    CONST robtarget T2024:=[[60.250034,78.904563,16.249831],[1.000000,0.000000,0.000000,0.000000],[0,0,-1,0],[9E+09,9E+09,9E+09,9E+09,9E+09,9E+09]];
    CONST robtarget T2025:=[[60.250034,32.487797,16.249831],[1.000000,0.000000,0.000000,0.000000],[0,0,-1,0],[9E+09,9E+09,9E+09,9E+09,9E+09,9E+09]];
    CONST robtarget T2026:=[[61.750040,32.676352,16.249831],[1.000000,0.000000,0.000000,0.000000],[0,0,-1,0],[9E+09,9E+09,9E+09,9E+09,9E+09,9E+09]];
    CONST robtarget T2027:=[[61.750040,78.498231,16.249831],[1.000000,0.000000,0.000000,0.000000],[0,0,-1,0],[9E+09,9E+09,9E+09,9E+09,9E+09,9E+09]];
    CONST robtarget T2028:=[[63.250046,77.962337,16.249831],[1.000000,0.000000,0.000000,0.000000],[0,0,-1,0],[9E+09,9E+09,9E+09,9E+09,9E+09,9E+09]];
    CONST robtarget T2029:=[[63.250046,32.936847,16.249831],[1.000000,0.000000,0.000000,0.000000],[0,0,-1,0],[9E+09,9E+09,9E+09,9E+09,9E+09,9E+09]];
    CONST robtarget T2030:=[[64.750052,33.276223,16.249831],[1.000000,0.000000,0.000000,0.000000],[0,0,-1,0],[9E+09,9E+09,9E+09,9E+09,9E+09,9E+09]];
    CONST robtarget T2031:=[[64.750052,77.237553,16.249831],[1.000000,0.000000,0.000000,0.000000],[0,0,-1,0],[9E+09,9E+09,9E+09,9E+09,9E+09,9E+09]];
    CONST robtarget T2032:=[[66.250058,76.248790,16.249831],[1.000000,0.000000,0.000000,0.000000],[0,0,-1,0],[9E+09,9E+09,9E+09,9E+09,9E+09,9E+09]];
    CONST robtarget T2033:=[[66.250058,33.701895,16.249831],[1.000000,0.000000,0.000000,0.000000],[0,0,-1,0],[9E+09,9E+09,9E+09,9E+09,9E+09,9E+09]];
    CONST robtarget T2034:=[[67.750064,34.280483,16.249831],[1.000000,0.000000,0.000000,0.000000],[0,0,-1,0],[9E+09,9E+09,9E+09,9E+09,9E+09,9E+09]];
    CONST robtarget T2035:=[[67.750064,74.766975,16.249831],[1.000000,0.000000,0.000000,0.000000],[0,0,-1,0],[9E+09,9E+09,9E+09,9E+09,9E+09,9E+09]];
    CONST robtarget T2036:=[[69.250070,72.779272,16.249831],[1.000000,0.000000,0.000000,0.000000],[0,0,-1,0],[9E+09,9E+09,9E+09,9E+09,9E+09,9E+09]];
    CONST robtarget T2037:=[[69.250070,34.893685,16.249831],[1.000000,0.000000,0.000000,0.000000],[0,0,-1,0],[9E+09,9E+09,9E+09,9E+09,9E+09,9E+09]];
    CONST robtarget T2038:=[[70.750076,35.855715,16.249831],[1.000000,0.000000,0.000000,0.000000],[0,0,-1,0],[9E+09,9E+09,9E+09,9E+09,9E+09,9E+09]];
    CONST robtarget T2039:=[[70.750076,70.592401,16.249831],[1.000000,0.000000,0.000000,0.000000],[0,0,-1,0],[9E+09,9E+09,9E+09,9E+09,9E+09,9E+09]];
    CONST robtarget T2040:=[[72.250082,71.487627,16.249831],[1.000000,0.000000,0.000000,0.000000],[0,0,-1,0],[9E+09,9E+09,9E+09,9E+09,9E+09,9E+09]];
    CONST robtarget T2041:=[[72.250082,36.807675,16.249831],[1.000000,0.000000,0.000000,0.000000],[0,0,-1,0],[9E+09,9E+09,9E+09,9E+09,9E+09,9E+09]];
    CONST robtarget T2042:=[[73.750088,38.399045,16.249831],[1.000000,0.000000,0.000000,0.000000],[0,0,-1,0],[9E+09,9E+09,9E+09,9E+09,9E+09,9E+09]];
    CONST robtarget T2043:=[[73.750088,70.448227,16.249831],[1.000000,0.000000,0.000000,0.000000],[0,0,-1,0],[9E+09,9E+09,9E+09,9E+09,9E+09,9E+09]];
    CONST robtarget T2044:=[[75.250094,67.768342,16.249831],[1.000000,0.000000,0.000000,0.000000],[0,0,-1,0],[9E+09,9E+09,9E+09,9E+09,9E+09,9E+09]];
    CONST robtarget T2045:=[[75.250094,40.369976,16.249831],[1.000000,0.000000,0.000000,0.000000],[0,0,-1,0],[9E+09,9E+09,9E+09,9E+09,9E+09,9E+09]];
    CONST robtarget T2046:=[[76.750100,43.140634,16.249831],[1.000000,0.000000,0.000000,0.000000],[0,0,-1,0],[9E+09,9E+09,9E+09,9E+09,9E+09,9E+09]];
    CONST robtarget T2047:=[[76.750100,63.221678,16.249831],[1.000000,0.000000,0.000000,0.000000],[0,0,-1,0],[9E+09,9E+09,9E+09,9E+09,9E+09,9E+09]];
    CONST robtarget T2048:=[[78.250106,56.651419,16.249831],[1.000000,0.000000,0.000000,0.000000],[0,0,-1,0],[9E+09,9E+09,9E+09,9E+09,9E+09,9E+09]];
    CONST robtarget T2049:=[[78.250106,48.862612,16.249831],[1.000000,0.000000,0.000000,0.000000],[0,0,-1,0],[9E+09,9E+09,9E+09,9E+09,9E+09,9E+09]];
    CONST robtarget T2050:=[[77.500103,48.233244,16.749841],[1.000000,0.000000,0.000000,0.000000],[0,0,-1,0],[9E+09,9E+09,9E+09,9E+09,9E+09,9E+09]];
    CONST robtarget T2051:=[[77.500103,59.623165,16.749841],[1.000000,0.000000,0.000000,0.000000],[0,0,-1,0],[9E+09,9E+09,9E+09,9E+09,9E+09,9E+09]];
    CONST robtarget T2052:=[[77.500103,48.233244,16.749841],[1.000000,0.000000,0.000000,0.000000],[0,0,-1,0],[9E+09,9E+09,9E+09,9E+09,9E+09,9E+09]];
    CONST robtarget T2053:=[[77.500103,59.623165,16.749841],[1.000000,0.000000,0.000000,0.000000],[0,0,-1,0],[9E+09,9E+09,9E+09,9E+09,9E+09,9E+09]];
    CONST robtarget T2054:=[[76.000097,65.184856,16.749841],[1.000000,0.000000,0.000000,0.000000],[0,0,-1,0],[9E+09,9E+09,9E+09,9E+09,9E+09,9E+09]];
    CONST robtarget T2055:=[[76.000097,41.932974,16.749841],[1.000000,0.000000,0.000000,0.000000],[0,0,-1,0],[9E+09,9E+09,9E+09,9E+09,9E+09,9E+09]];
    CONST robtarget T2056:=[[74.500091,39.400333,16.749841],[1.000000,0.000000,0.000000,0.000000],[0,0,-1,0],[9E+09,9E+09,9E+09,9E+09,9E+09,9E+09]];
    CONST robtarget T2057:=[[74.500091,69.124433,16.749841],[1.000000,0.000000,0.000000,0.000000],[0,0,-1,0],[9E+09,9E+09,9E+09,9E+09,9E+09,9E+09]];
    CONST robtarget T2058:=[[73.000085,71.338605,16.749841],[1.000000,0.000000,0.000000,0.000000],[0,0,-1,0],[9E+09,9E+09,9E+09,9E+09,9E+09,9E+09]];
    CONST robtarget T2059:=[[73.000085,37.732430,16.749841],[1.000000,0.000000,0.000000,0.000000],[0,0,-1,0],[9E+09,9E+09,9E+09,9E+09,9E+09,9E+09]];
    CONST robtarget T2060:=[[71.500079,36.421505,16.749841],[1.000000,0.000000,0.000000,0.000000],[0,0,-1,0],[9E+09,9E+09,9E+09,9E+09,9E+09,9E+09]];
    CONST robtarget T2061:=[[71.500079,70.991778,16.749841],[1.000000,0.000000,0.000000,0.000000],[0,0,-1,0],[9E+09,9E+09,9E+09,9E+09,9E+09,9E+09]];
    CONST robtarget T2062:=[[70.000073,71.577935,16.749841],[1.000000,0.000000,0.000000,0.000000],[0,0,-1,0],[9E+09,9E+09,9E+09,9E+09,9E+09,9E+09]];
    CONST robtarget T2063:=[[70.000073,35.459476,16.749841],[1.000000,0.000000,0.000000,0.000000],[0,0,-1,0],[9E+09,9E+09,9E+09,9E+09,9E+09,9E+09]];
    CONST robtarget T2064:=[[68.500067,34.636854,16.749841],[1.000000,0.000000,0.000000,0.000000],[0,0,-1,0],[9E+09,9E+09,9E+09,9E+09,9E+09,9E+09]];
    CONST robtarget T2065:=[[68.500067,73.714208,16.749841],[1.000000,0.000000,0.000000,0.000000],[0,0,-1,0],[9E+09,9E+09,9E+09,9E+09,9E+09,9E+09]];
    CONST robtarget T2066:=[[67.000061,75.529975,16.749841],[1.000000,0.000000,0.000000,0.000000],[0,0,-1,0],[9E+09,9E+09,9E+09,9E+09,9E+09,9E+09]];
    CONST robtarget T2067:=[[67.000061,34.067929,16.749841],[1.000000,0.000000,0.000000,0.000000],[0,0,-1,0],[9E+09,9E+09,9E+09,9E+09,9E+09,9E+09]];
    CONST robtarget T2068:=[[65.500055,33.523693,16.749841],[1.000000,0.000000,0.000000,0.000000],[0,0,-1,0],[9E+09,9E+09,9E+09,9E+09,9E+09,9E+09]];
    CONST robtarget T2069:=[[65.500055,76.783651,16.749841],[1.000000,0.000000,0.000000,0.000000],[0,0,-1,0],[9E+09,9E+09,9E+09,9E+09,9E+09,9E+09]];
    CONST robtarget T2070:=[[64.000049,77.607482,16.749841],[1.000000,0.000000,0.000000,0.000000],[0,0,-1,0],[9E+09,9E+09,9E+09,9E+09,9E+09,9E+09]];
    CONST robtarget T2071:=[[64.000049,33.181966,16.749841],[1.000000,0.000000,0.000000,0.000000],[0,0,-1,0],[9E+09,9E+09,9E+09,9E+09,9E+09,9E+09]];
    CONST robtarget T2072:=[[62.500043,32.845958,16.749841],[1.000000,0.000000,0.000000,0.000000],[0,0,-1,0],[9E+09,9E+09,9E+09,9E+09,9E+09,9E+09]];
    CONST robtarget T2073:=[[62.500043,78.210676,16.749841],[1.000000,0.000000,0.000000,0.000000],[0,0,-1,0],[9E+09,9E+09,9E+09,9E+09,9E+09,9E+09]];
    CONST robtarget T2074:=[[61.000037,78.726702,16.749841],[1.000000,0.000000,0.000000,0.000000],[0,0,-1,0],[9E+09,9E+09,9E+09,9E+09,9E+09,9E+09]];
    CONST robtarget T2075:=[[61.000037,32.654827,16.749841],[1.000000,0.000000,0.000000,0.000000],[0,0,-1,0],[9E+09,9E+09,9E+09,9E+09,9E+09,9E+09]];
    CONST robtarget T2076:=[[59.500031,32.472908,16.749841],[1.000000,0.000000,0.000000,0.000000],[0,0,-1,0],[9E+09,9E+09,9E+09,9E+09,9E+09,9E+09]];
    CONST robtarget T2077:=[[59.500031,79.071134,16.749841],[1.000000,0.000000,0.000000,0.000000],[0,0,-1,0],[9E+09,9E+09,9E+09,9E+09,9E+09,9E+09]];
    CONST robtarget T2078:=[[58.000025,79.360542,16.749841],[1.000000,0.000000,0.000000,0.000000],[0,0,-1,0],[9E+09,9E+09,9E+09,9E+09,9E+09,9E+09]];
    CONST robtarget T2079:=[[58.000025,32.352211,16.749841],[1.000000,0.000000,0.000000,0.000000],[0,0,-1,0],[9E+09,9E+09,9E+09,9E+09,9E+09,9E+09]];
    CONST robtarget T2080:=[[56.500019,32.279634,16.749841],[1.000000,0.000000,0.000000,0.000000],[0,0,-1,0],[9E+09,9E+09,9E+09,9E+09,9E+09,9E+09]];
    CONST robtarget T2081:=[[56.500019,79.716007,16.749841],[1.000000,0.000000,0.000000,0.000000],[0,0,-1,0],[9E+09,9E+09,9E+09,9E+09,9E+09,9E+09]];
    CONST robtarget T2082:=[[55.000013,79.976085,16.749841],[1.000000,0.000000,0.000000,0.000000],[0,0,-1,0],[9E+09,9E+09,9E+09,9E+09,9E+09,9E+09]];
    CONST robtarget T2083:=[[55.000013,32.242406,16.749841],[1.000000,0.000000,0.000000,0.000000],[0,0,-1,0],[9E+09,9E+09,9E+09,9E+09,9E+09,9E+09]];
    CONST robtarget T2084:=[[53.500007,32.279634,16.749841],[1.000000,0.000000,0.000000,0.000000],[0,0,-1,0],[9E+09,9E+09,9E+09,9E+09,9E+09,9E+09]];
    CONST robtarget T2085:=[[53.500007,79.716007,16.749841],[1.000000,0.000000,0.000000,0.000000],[0,0,-1,0],[9E+09,9E+09,9E+09,9E+09,9E+09,9E+09]];
    CONST robtarget T2086:=[[52.000001,79.360541,16.749841],[1.000000,0.000000,0.000000,0.000000],[0,0,-1,0],[9E+09,9E+09,9E+09,9E+09,9E+09,9E+09]];
    CONST robtarget T2087:=[[52.000001,32.352210,16.749841],[1.000000,0.000000,0.000000,0.000000],[0,0,-1,0],[9E+09,9E+09,9E+09,9E+09,9E+09,9E+09]];
    CONST robtarget T2088:=[[50.499995,32.472907,16.749841],[1.000000,0.000000,0.000000,0.000000],[0,0,-1,0],[9E+09,9E+09,9E+09,9E+09,9E+09,9E+09]];
    CONST robtarget T2089:=[[50.499995,79.071135,16.749841],[1.000000,0.000000,0.000000,0.000000],[0,0,-1,0],[9E+09,9E+09,9E+09,9E+09,9E+09,9E+09]];
    CONST robtarget T2090:=[[48.999989,78.726701,16.749841],[1.000000,0.000000,0.000000,0.000000],[0,0,-1,0],[9E+09,9E+09,9E+09,9E+09,9E+09,9E+09]];
    CONST robtarget T2091:=[[48.999989,32.654826,16.749841],[1.000000,0.000000,0.000000,0.000000],[0,0,-1,0],[9E+09,9E+09,9E+09,9E+09,9E+09,9E+09]];
    CONST robtarget T2092:=[[47.499983,32.845957,16.749841],[1.000000,0.000000,0.000000,0.000000],[0,0,-1,0],[9E+09,9E+09,9E+09,9E+09,9E+09,9E+09]];
    CONST robtarget T2093:=[[47.499983,78.210668,16.749841],[1.000000,0.000000,0.000000,0.000000],[0,0,-1,0],[9E+09,9E+09,9E+09,9E+09,9E+09,9E+09]];
    CONST robtarget T2094:=[[45.999977,77.607480,16.749841],[1.000000,0.000000,0.000000,0.000000],[0,0,-1,0],[9E+09,9E+09,9E+09,9E+09,9E+09,9E+09]];
    CONST robtarget T2095:=[[45.999977,33.181963,16.749841],[1.000000,0.000000,0.000000,0.000000],[0,0,-1,0],[9E+09,9E+09,9E+09,9E+09,9E+09,9E+09]];
    CONST robtarget T2096:=[[44.499971,33.523691,16.749841],[1.000000,0.000000,0.000000,0.000000],[0,0,-1,0],[9E+09,9E+09,9E+09,9E+09,9E+09,9E+09]];
    CONST robtarget T2097:=[[44.499971,76.783660,16.749841],[1.000000,0.000000,0.000000,0.000000],[0,0,-1,0],[9E+09,9E+09,9E+09,9E+09,9E+09,9E+09]];
    CONST robtarget T2098:=[[42.999965,75.529990,16.749841],[1.000000,0.000000,0.000000,0.000000],[0,0,-1,0],[9E+09,9E+09,9E+09,9E+09,9E+09,9E+09]];
    CONST robtarget T2099:=[[42.999965,34.067925,16.749841],[1.000000,0.000000,0.000000,0.000000],[0,0,-1,0],[9E+09,9E+09,9E+09,9E+09,9E+09,9E+09]];
    CONST robtarget T2100:=[[41.499959,34.636849,16.749841],[1.000000,0.000000,0.000000,0.000000],[0,0,-1,0],[9E+09,9E+09,9E+09,9E+09,9E+09,9E+09]];
    CONST robtarget T2101:=[[41.499959,73.714226,16.749841],[1.000000,0.000000,0.000000,0.000000],[0,0,-1,0],[9E+09,9E+09,9E+09,9E+09,9E+09,9E+09]];
    CONST robtarget T2102:=[[39.999953,71.577955,16.749841],[1.000000,0.000000,0.000000,0.000000],[0,0,-1,0],[9E+09,9E+09,9E+09,9E+09,9E+09,9E+09]];
    CONST robtarget T2103:=[[39.999953,35.459468,16.749841],[1.000000,0.000000,0.000000,0.000000],[0,0,-1,0],[9E+09,9E+09,9E+09,9E+09,9E+09,9E+09]];
    CONST robtarget T2104:=[[38.499947,36.421498,16.749841],[1.000000,0.000000,0.000000,0.000000],[0,0,-1,0],[9E+09,9E+09,9E+09,9E+09,9E+09,9E+09]];
    CONST robtarget T2105:=[[38.499947,70.991724,16.749841],[1.000000,0.000000,0.000000,0.000000],[0,0,-1,0],[9E+09,9E+09,9E+09,9E+09,9E+09,9E+09]];
    CONST robtarget T2106:=[[36.999941,71.338623,16.749841],[1.000000,0.000000,0.000000,0.000000],[0,0,-1,0],[9E+09,9E+09,9E+09,9E+09,9E+09,9E+09]];
    CONST robtarget T2107:=[[36.999941,37.732418,16.749841],[1.000000,0.000000,0.000000,0.000000],[0,0,-1,0],[9E+09,9E+09,9E+09,9E+09,9E+09,9E+09]];
    CONST robtarget T2108:=[[35.499935,39.400322,16.749841],[1.000000,0.000000,0.000000,0.000000],[0,0,-1,0],[9E+09,9E+09,9E+09,9E+09,9E+09,9E+09]];
    CONST robtarget T2109:=[[35.499935,69.123986,16.749841],[1.000000,0.000000,0.000000,0.000000],[0,0,-1,0],[9E+09,9E+09,9E+09,9E+09,9E+09,9E+09]];
    CONST robtarget T2110:=[[33.999929,65.171816,16.749841],[1.000000,0.000000,0.000000,0.000000],[0,0,-1,0],[9E+09,9E+09,9E+09,9E+09,9E+09,9E+09]];
    CONST robtarget T2111:=[[33.999929,41.932953,16.749841],[1.000000,0.000000,0.000000,0.000000],[0,0,-1,0],[9E+09,9E+09,9E+09,9E+09,9E+09,9E+09]];
    CONST robtarget T2112:=[[32.499923,48.233209,16.749841],[1.000000,0.000000,0.000000,0.000000],[0,0,-1,0],[9E+09,9E+09,9E+09,9E+09,9E+09,9E+09]];
    CONST robtarget T2113:=[[32.499923,59.589242,16.749841],[1.000000,0.000000,0.000000,0.000000],[0,0,-1,0],[9E+09,9E+09,9E+09,9E+09,9E+09,9E+09]];
    CONST robtarget T2114:=[[32.500647,49.771236,17.249851],[1.000000,0.000000,0.000000,0.000000],[0,0,-1,0],[9E+09,9E+09,9E+09,9E+09,9E+09,9E+09]];
    CONST robtarget T2115:=[[32.500647,58.735329,17.249851],[1.000000,0.000000,0.000000,0.000000],[0,0,-1,0],[9E+09,9E+09,9E+09,9E+09,9E+09,9E+09]];
    CONST robtarget T2116:=[[32.500647,49.771236,17.249851],[1.000000,0.000000,0.000000,0.000000],[0,0,-1,0],[9E+09,9E+09,9E+09,9E+09,9E+09,9E+09]];
    CONST robtarget T2117:=[[32.500647,58.735329,17.249851],[1.000000,0.000000,0.000000,0.000000],[0,0,-1,0],[9E+09,9E+09,9E+09,9E+09,9E+09,9E+09]];
    CONST robtarget T2118:=[[34.000653,64.598612,17.249851],[1.000000,0.000000,0.000000,0.000000],[0,0,-1,0],[9E+09,9E+09,9E+09,9E+09,9E+09,9E+09]];
    CONST robtarget T2119:=[[34.000653,42.603949,17.249851],[1.000000,0.000000,0.000000,0.000000],[0,0,-1,0],[9E+09,9E+09,9E+09,9E+09,9E+09,9E+09]];
    CONST robtarget T2120:=[[35.500659,39.775888,17.249851],[1.000000,0.000000,0.000000,0.000000],[0,0,-1,0],[9E+09,9E+09,9E+09,9E+09,9E+09,9E+09]];
    CONST robtarget T2121:=[[35.500659,68.767657,17.249851],[1.000000,0.000000,0.000000,0.000000],[0,0,-1,0],[9E+09,9E+09,9E+09,9E+09,9E+09,9E+09]];
    CONST robtarget T2122:=[[37.000665,71.349106,17.249851],[1.000000,0.000000,0.000000,0.000000],[0,0,-1,0],[9E+09,9E+09,9E+09,9E+09,9E+09,9E+09]];
    CONST robtarget T2123:=[[37.000665,37.988033,17.249851],[1.000000,0.000000,0.000000,0.000000],[0,0,-1,0],[9E+09,9E+09,9E+09,9E+09,9E+09,9E+09]];
    CONST robtarget T2124:=[[38.500671,36.525985,17.249851],[1.000000,0.000000,0.000000,0.000000],[0,0,-1,0],[9E+09,9E+09,9E+09,9E+09,9E+09,9E+09]];
    CONST robtarget T2125:=[[38.500671,71.602983,17.249851],[1.000000,0.000000,0.000000,0.000000],[0,0,-1,0],[9E+09,9E+09,9E+09,9E+09,9E+09,9E+09]];
    CONST robtarget T2126:=[[40.000677,71.445291,17.249851],[1.000000,0.000000,0.000000,0.000000],[0,0,-1,0],[9E+09,9E+09,9E+09,9E+09,9E+09,9E+09]];
    CONST robtarget T2127:=[[40.000677,35.545486,17.249851],[1.000000,0.000000,0.000000,0.000000],[0,0,-1,0],[9E+09,9E+09,9E+09,9E+09,9E+09,9E+09]];
    CONST robtarget T2128:=[[41.500683,34.708483,17.249851],[1.000000,0.000000,0.000000,0.000000],[0,0,-1,0],[9E+09,9E+09,9E+09,9E+09,9E+09,9E+09]];
    CONST robtarget T2129:=[[41.500683,73.587282,17.249851],[1.000000,0.000000,0.000000,0.000000],[0,0,-1,0],[9E+09,9E+09,9E+09,9E+09,9E+09,9E+09]];
    CONST robtarget T2130:=[[43.000689,75.445051,17.249851],[1.000000,0.000000,0.000000,0.000000],[0,0,-1,0],[9E+09,9E+09,9E+09,9E+09,9E+09,9E+09]];
    CONST robtarget T2131:=[[43.000689,34.139559,17.249851],[1.000000,0.000000,0.000000,0.000000],[0,0,-1,0],[9E+09,9E+09,9E+09,9E+09,9E+09,9E+09]];
    CONST robtarget T2132:=[[44.500695,33.596928,17.249851],[1.000000,0.000000,0.000000,0.000000],[0,0,-1,0],[9E+09,9E+09,9E+09,9E+09,9E+09,9E+09]];
    CONST robtarget T2133:=[[44.500695,76.747362,17.249851],[1.000000,0.000000,0.000000,0.000000],[0,0,-1,0],[9E+09,9E+09,9E+09,9E+09,9E+09,9E+09]];
    CONST robtarget T2134:=[[46.000701,77.591605,17.249851],[1.000000,0.000000,0.000000,0.000000],[0,0,-1,0],[9E+09,9E+09,9E+09,9E+09,9E+09,9E+09]];
    CONST robtarget T2135:=[[46.000701,33.258335,17.249851],[1.000000,0.000000,0.000000,0.000000],[0,0,-1,0],[9E+09,9E+09,9E+09,9E+09,9E+09,9E+09]];
    CONST robtarget T2136:=[[47.500707,32.921166,17.249851],[1.000000,0.000000,0.000000,0.000000],[0,0,-1,0],[9E+09,9E+09,9E+09,9E+09,9E+09,9E+09]];
    CONST robtarget T2137:=[[47.500707,78.204680,17.249851],[1.000000,0.000000,0.000000,0.000000],[0,0,-1,0],[9E+09,9E+09,9E+09,9E+09,9E+09,9E+09]];
    CONST robtarget T2138:=[[49.000713,78.722227,17.249851],[1.000000,0.000000,0.000000,0.000000],[0,0,-1,0],[9E+09,9E+09,9E+09,9E+09,9E+09,9E+09]];
    CONST robtarget T2139:=[[49.000713,32.728774,17.249851],[1.000000,0.000000,0.000000,0.000000],[0,0,-1,0],[9E+09,9E+09,9E+09,9E+09,9E+09,9E+09]];
    CONST robtarget T2140:=[[50.500719,32.544623,17.249851],[1.000000,0.000000,0.000000,0.000000],[0,0,-1,0],[9E+09,9E+09,9E+09,9E+09,9E+09,9E+09]];
    CONST robtarget T2141:=[[50.500719,79.065689,17.249851],[1.000000,0.000000,0.000000,0.000000],[0,0,-1,0],[9E+09,9E+09,9E+09,9E+09,9E+09,9E+09]];
    CONST robtarget T2142:=[[52.000725,79.353294,17.249851],[1.000000,0.000000,0.000000,0.000000],[0,0,-1,0],[9E+09,9E+09,9E+09,9E+09,9E+09,9E+09]];
    CONST robtarget T2143:=[[52.000725,32.425930,17.249851],[1.000000,0.000000,0.000000,0.000000],[0,0,-1,0],[9E+09,9E+09,9E+09,9E+09,9E+09,9E+09]];
    CONST robtarget T2144:=[[53.500731,32.352404,17.249851],[1.000000,0.000000,0.000000,0.000000],[0,0,-1,0],[9E+09,9E+09,9E+09,9E+09,9E+09,9E+09]];
    CONST robtarget T2145:=[[53.500731,79.707174,17.249851],[1.000000,0.000000,0.000000,0.000000],[0,0,-1,0],[9E+09,9E+09,9E+09,9E+09,9E+09,9E+09]];
    CONST robtarget T2146:=[[55.000737,79.961091,17.249851],[1.000000,0.000000,0.000000,0.000000],[0,0,-1,0],[9E+09,9E+09,9E+09,9E+09,9E+09,9E+09]];
    CONST robtarget T2147:=[[55.000737,32.319476,17.249851],[1.000000,0.000000,0.000000,0.000000],[0,0,-1,0],[9E+09,9E+09,9E+09,9E+09,9E+09,9E+09]];
    CONST robtarget T2148:=[[56.500743,32.352427,17.249851],[1.000000,0.000000,0.000000,0.000000],[0,0,-1,0],[9E+09,9E+09,9E+09,9E+09,9E+09,9E+09]];
    CONST robtarget T2149:=[[56.500743,79.706797,17.249851],[1.000000,0.000000,0.000000,0.000000],[0,0,-1,0],[9E+09,9E+09,9E+09,9E+09,9E+09,9E+09]];
    CONST robtarget T2150:=[[58.000749,79.353018,17.249851],[1.000000,0.000000,0.000000,0.000000],[0,0,-1,0],[9E+09,9E+09,9E+09,9E+09,9E+09,9E+09]];
    CONST robtarget T2151:=[[58.000749,32.426042,17.249851],[1.000000,0.000000,0.000000,0.000000],[0,0,-1,0],[9E+09,9E+09,9E+09,9E+09,9E+09,9E+09]];
    CONST robtarget T2152:=[[59.500755,32.544745,17.249851],[1.000000,0.000000,0.000000,0.000000],[0,0,-1,0],[9E+09,9E+09,9E+09,9E+09,9E+09,9E+09]];
    CONST robtarget T2153:=[[59.500755,79.065362,17.249851],[1.000000,0.000000,0.000000,0.000000],[0,0,-1,0],[9E+09,9E+09,9E+09,9E+09,9E+09,9E+09]];
    CONST robtarget T2154:=[[61.000761,78.721895,17.249851],[1.000000,0.000000,0.000000,0.000000],[0,0,-1,0],[9E+09,9E+09,9E+09,9E+09,9E+09,9E+09]];
    CONST robtarget T2155:=[[61.000761,32.728961,17.249851],[1.000000,0.000000,0.000000,0.000000],[0,0,-1,0],[9E+09,9E+09,9E+09,9E+09,9E+09,9E+09]];
    CONST robtarget T2156:=[[62.500767,32.921494,17.249851],[1.000000,0.000000,0.000000,0.000000],[0,0,-1,0],[9E+09,9E+09,9E+09,9E+09,9E+09,9E+09]];
    CONST robtarget T2157:=[[62.500767,78.204203,17.249851],[1.000000,0.000000,0.000000,0.000000],[0,0,-1,0],[9E+09,9E+09,9E+09,9E+09,9E+09,9E+09]];
    CONST robtarget T2158:=[[64.000773,77.590903,17.249851],[1.000000,0.000000,0.000000,0.000000],[0,0,-1,0],[9E+09,9E+09,9E+09,9E+09,9E+09,9E+09]];
    CONST robtarget T2159:=[[64.000773,33.258663,17.249851],[1.000000,0.000000,0.000000,0.000000],[0,0,-1,0],[9E+09,9E+09,9E+09,9E+09,9E+09,9E+09]];
    CONST robtarget T2160:=[[65.500779,33.597267,17.249851],[1.000000,0.000000,0.000000,0.000000],[0,0,-1,0],[9E+09,9E+09,9E+09,9E+09,9E+09,9E+09]];
    CONST robtarget T2161:=[[65.500779,76.746249,17.249851],[1.000000,0.000000,0.000000,0.000000],[0,0,-1,0],[9E+09,9E+09,9E+09,9E+09,9E+09,9E+09]];
    CONST robtarget T2162:=[[67.000785,75.443377,17.249851],[1.000000,0.000000,0.000000,0.000000],[0,0,-1,0],[9E+09,9E+09,9E+09,9E+09,9E+09,9E+09]];
    CONST robtarget T2163:=[[67.000785,34.140112,17.249851],[1.000000,0.000000,0.000000,0.000000],[0,0,-1,0],[9E+09,9E+09,9E+09,9E+09,9E+09,9E+09]];
    CONST robtarget T2164:=[[68.500791,34.709037,17.249851],[1.000000,0.000000,0.000000,0.000000],[0,0,-1,0],[9E+09,9E+09,9E+09,9E+09,9E+09,9E+09]];
    CONST robtarget T2165:=[[68.500791,73.585211,17.249851],[1.000000,0.000000,0.000000,0.000000],[0,0,-1,0],[9E+09,9E+09,9E+09,9E+09,9E+09,9E+09]];
    CONST robtarget T2166:=[[70.000797,71.443139,17.249851],[1.000000,0.000000,0.000000,0.000000],[0,0,-1,0],[9E+09,9E+09,9E+09,9E+09,9E+09,9E+09]];
    CONST robtarget T2167:=[[70.000797,35.546440,17.249851],[1.000000,0.000000,0.000000,0.000000],[0,0,-1,0],[9E+09,9E+09,9E+09,9E+09,9E+09,9E+09]];
    CONST robtarget T2168:=[[71.500803,36.526939,17.249851],[1.000000,0.000000,0.000000,0.000000],[0,0,-1,0],[9E+09,9E+09,9E+09,9E+09,9E+09,9E+09]];
    CONST robtarget T2169:=[[71.500803,71.604118,17.249851],[1.000000,0.000000,0.000000,0.000000],[0,0,-1,0],[9E+09,9E+09,9E+09,9E+09,9E+09,9E+09]];
    CONST robtarget T2170:=[[73.000809,71.347501,17.249851],[1.000000,0.000000,0.000000,0.000000],[0,0,-1,0],[9E+09,9E+09,9E+09,9E+09,9E+09,9E+09]];
    CONST robtarget T2171:=[[73.000809,37.989734,17.249851],[1.000000,0.000000,0.000000,0.000000],[0,0,-1,0],[9E+09,9E+09,9E+09,9E+09,9E+09,9E+09]];
    CONST robtarget T2172:=[[74.500815,39.778551,17.249851],[1.000000,0.000000,0.000000,0.000000],[0,0,-1,0],[9E+09,9E+09,9E+09,9E+09,9E+09,9E+09]];
    CONST robtarget T2173:=[[74.500815,68.766048,17.249851],[1.000000,0.000000,0.000000,0.000000],[0,0,-1,0],[9E+09,9E+09,9E+09,9E+09,9E+09,9E+09]];
    CONST robtarget T2174:=[[76.000821,64.618344,17.249851],[1.000000,0.000000,0.000000,0.000000],[0,0,-1,0],[9E+09,9E+09,9E+09,9E+09,9E+09,9E+09]];
    CONST robtarget T2175:=[[76.000821,42.607408,17.249851],[1.000000,0.000000,0.000000,0.000000],[0,0,-1,0],[9E+09,9E+09,9E+09,9E+09,9E+09,9E+09]];
    CONST robtarget T2176:=[[77.500827,49.776972,17.249851],[1.000000,0.000000,0.000000,0.000000],[0,0,-1,0],[9E+09,9E+09,9E+09,9E+09,9E+09,9E+09]];
    CONST robtarget T2177:=[[77.500827,58.775319,17.249851],[1.000000,0.000000,0.000000,0.000000],[0,0,-1,0],[9E+09,9E+09,9E+09,9E+09,9E+09,9E+09]];
    CONST robtarget T2178:=[[76.750757,48.951712,17.749861],[1.000000,0.000000,0.000000,0.000000],[0,0,-1,0],[9E+09,9E+09,9E+09,9E+09,9E+09,9E+09]];
    CONST robtarget T2179:=[[76.750757,61.091970,17.749861],[1.000000,0.000000,0.000000,0.000000],[0,0,-1,0],[9E+09,9E+09,9E+09,9E+09,9E+09,9E+09]];
    CONST robtarget T2180:=[[76.750757,48.951712,17.749861],[1.000000,0.000000,0.000000,0.000000],[0,0,-1,0],[9E+09,9E+09,9E+09,9E+09,9E+09,9E+09]];
    CONST robtarget T2181:=[[76.750757,61.091970,17.749861],[1.000000,0.000000,0.000000,0.000000],[0,0,-1,0],[9E+09,9E+09,9E+09,9E+09,9E+09,9E+09]];
    CONST robtarget T2182:=[[75.250751,66.389476,17.749861],[1.000000,0.000000,0.000000,0.000000],[0,0,-1,0],[9E+09,9E+09,9E+09,9E+09,9E+09,9E+09]];
    CONST robtarget T2183:=[[75.250751,41.731543,17.749861],[1.000000,0.000000,0.000000,0.000000],[0,0,-1,0],[9E+09,9E+09,9E+09,9E+09,9E+09,9E+09]];
    CONST robtarget T2184:=[[73.750745,39.279875,17.749861],[1.000000,0.000000,0.000000,0.000000],[0,0,-1,0],[9E+09,9E+09,9E+09,9E+09,9E+09,9E+09]];
    CONST robtarget T2185:=[[73.750745,70.036081,17.749861],[1.000000,0.000000,0.000000,0.000000],[0,0,-1,0],[9E+09,9E+09,9E+09,9E+09,9E+09,9E+09]];
    CONST robtarget T2186:=[[72.250739,71.928438,17.749861],[1.000000,0.000000,0.000000,0.000000],[0,0,-1,0],[9E+09,9E+09,9E+09,9E+09,9E+09,9E+09]];
    CONST robtarget T2187:=[[72.250739,37.527051,17.749861],[1.000000,0.000000,0.000000,0.000000],[0,0,-1,0],[9E+09,9E+09,9E+09,9E+09,9E+09,9E+09]];
    CONST robtarget T2188:=[[70.750733,36.288030,17.749861],[1.000000,0.000000,0.000000,0.000000],[0,0,-1,0],[9E+09,9E+09,9E+09,9E+09,9E+09,9E+09]];
    CONST robtarget T2189:=[[70.750733,70.255536,17.749861],[1.000000,0.000000,0.000000,0.000000],[0,0,-1,0],[9E+09,9E+09,9E+09,9E+09,9E+09,9E+09]];
    CONST robtarget T2190:=[[69.250727,72.414526,17.749861],[1.000000,0.000000,0.000000,0.000000],[0,0,-1,0],[9E+09,9E+09,9E+09,9E+09,9E+09,9E+09]];
    CONST robtarget T2191:=[[69.250727,35.307531,17.749861],[1.000000,0.000000,0.000000,0.000000],[0,0,-1,0],[9E+09,9E+09,9E+09,9E+09,9E+09,9E+09]];
    CONST robtarget T2192:=[[67.750721,34.588920,17.749861],[1.000000,0.000000,0.000000,0.000000],[0,0,-1,0],[9E+09,9E+09,9E+09,9E+09,9E+09,9E+09]];
    CONST robtarget T2193:=[[67.750721,74.507020,17.749861],[1.000000,0.000000,0.000000,0.000000],[0,0,-1,0],[9E+09,9E+09,9E+09,9E+09,9E+09,9E+09]];
    CONST robtarget T2194:=[[66.250715,76.132732,17.749861],[1.000000,0.000000,0.000000,0.000000],[0,0,-1,0],[9E+09,9E+09,9E+09,9E+09,9E+09,9E+09]];
    CONST robtarget T2195:=[[66.250715,33.964244,17.749861],[1.000000,0.000000,0.000000,0.000000],[0,0,-1,0],[9E+09,9E+09,9E+09,9E+09,9E+09,9E+09]];
    CONST robtarget T2196:=[[64.750709,33.503767,17.749861],[1.000000,0.000000,0.000000,0.000000],[0,0,-1,0],[9E+09,9E+09,9E+09,9E+09,9E+09,9E+09]];
    CONST robtarget T2197:=[[64.750709,77.200806,17.749861],[1.000000,0.000000,0.000000,0.000000],[0,0,-1,0],[9E+09,9E+09,9E+09,9E+09,9E+09,9E+09]];
    CONST robtarget T2198:=[[63.250703,77.939066,17.749861],[1.000000,0.000000,0.000000,0.000000],[0,0,-1,0],[9E+09,9E+09,9E+09,9E+09,9E+09,9E+09]];
    CONST robtarget T2199:=[[63.250703,33.166598,17.749861],[1.000000,0.000000,0.000000,0.000000],[0,0,-1,0],[9E+09,9E+09,9E+09,9E+09,9E+09,9E+09]];
    CONST robtarget T2200:=[[61.750697,32.898559,17.749861],[1.000000,0.000000,0.000000,0.000000],[0,0,-1,0],[9E+09,9E+09,9E+09,9E+09,9E+09,9E+09]];
    CONST robtarget T2201:=[[61.750697,78.458695,17.749861],[1.000000,0.000000,0.000000,0.000000],[0,0,-1,0],[9E+09,9E+09,9E+09,9E+09,9E+09,9E+09]];
    CONST robtarget T2202:=[[60.250691,78.890491,17.749861],[1.000000,0.000000,0.000000,0.000000],[0,0,-1,0],[9E+09,9E+09,9E+09,9E+09,9E+09,9E+09]];
    CONST robtarget T2203:=[[60.250691,32.707428,17.749861],[1.000000,0.000000,0.000000,0.000000],[0,0,-1,0],[9E+09,9E+09,9E+09,9E+09,9E+09,9E+09]];
    CONST robtarget T2204:=[[58.750685,32.557429,17.749861],[1.000000,0.000000,0.000000,0.000000],[0,0,-1,0],[9E+09,9E+09,9E+09,9E+09,9E+09,9E+09]];
    CONST robtarget T2205:=[[58.750685,79.208772,17.749861],[1.000000,0.000000,0.000000,0.000000],[0,0,-1,0],[9E+09,9E+09,9E+09,9E+09,9E+09,9E+09]];
    CONST robtarget T2206:=[[57.250679,79.501585,17.749861],[1.000000,0.000000,0.000000,0.000000],[0,0,-1,0],[9E+09,9E+09,9E+09,9E+09,9E+09,9E+09]];
    CONST robtarget T2207:=[[57.250679,32.442195,17.749861],[1.000000,0.000000,0.000000,0.000000],[0,0,-1,0],[9E+09,9E+09,9E+09,9E+09,9E+09,9E+09]];
    CONST robtarget T2208:=[[55.750673,32.413746,17.749861],[1.000000,0.000000,0.000000,0.000000],[0,0,-1,0],[9E+09,9E+09,9E+09,9E+09,9E+09,9E+09]];
    CONST robtarget T2209:=[[55.750673,79.831179,17.749861],[1.000000,0.000000,0.000000,0.000000],[0,0,-1,0],[9E+09,9E+09,9E+09,9E+09,9E+09,9E+09]];
    CONST robtarget T2210:=[[54.250667,79.831346,17.749861],[1.000000,0.000000,0.000000,0.000000],[0,0,-1,0],[9E+09,9E+09,9E+09,9E+09,9E+09,9E+09]];
    CONST robtarget T2211:=[[54.250667,32.413726,17.749861],[1.000000,0.000000,0.000000,0.000000],[0,0,-1,0],[9E+09,9E+09,9E+09,9E+09,9E+09,9E+09]];
    CONST robtarget T2212:=[[52.750661,32.442094,17.749861],[1.000000,0.000000,0.000000,0.000000],[0,0,-1,0],[9E+09,9E+09,9E+09,9E+09,9E+09,9E+09]];
    CONST robtarget T2213:=[[52.750661,79.501925,17.749861],[1.000000,0.000000,0.000000,0.000000],[0,0,-1,0],[9E+09,9E+09,9E+09,9E+09,9E+09,9E+09]];
    CONST robtarget T2214:=[[51.250655,79.208998,17.749861],[1.000000,0.000000,0.000000,0.000000],[0,0,-1,0],[9E+09,9E+09,9E+09,9E+09,9E+09,9E+09]];
    CONST robtarget T2215:=[[51.250655,32.557327,17.749861],[1.000000,0.000000,0.000000,0.000000],[0,0,-1,0],[9E+09,9E+09,9E+09,9E+09,9E+09,9E+09]];
    CONST robtarget T2216:=[[49.750649,32.707259,17.749861],[1.000000,0.000000,0.000000,0.000000],[0,0,-1,0],[9E+09,9E+09,9E+09,9E+09,9E+09,9E+09]];
    CONST robtarget T2217:=[[49.750649,78.890791,17.749861],[1.000000,0.000000,0.000000,0.000000],[0,0,-1,0],[9E+09,9E+09,9E+09,9E+09,9E+09,9E+09]];
    CONST robtarget T2218:=[[48.250643,78.459170,17.749861],[1.000000,0.000000,0.000000,0.000000],[0,0,-1,0],[9E+09,9E+09,9E+09,9E+09,9E+09,9E+09]];
    CONST robtarget T2219:=[[48.250643,32.898390,17.749861],[1.000000,0.000000,0.000000,0.000000],[0,0,-1,0],[9E+09,9E+09,9E+09,9E+09,9E+09,9E+09]];
    CONST robtarget T2220:=[[46.750637,33.166300,17.749861],[1.000000,0.000000,0.000000,0.000000],[0,0,-1,0],[9E+09,9E+09,9E+09,9E+09,9E+09,9E+09]];
    CONST robtarget T2221:=[[46.750637,77.939698,17.749861],[1.000000,0.000000,0.000000,0.000000],[0,0,-1,0],[9E+09,9E+09,9E+09,9E+09,9E+09,9E+09]];
    CONST robtarget T2222:=[[45.250631,77.201488,17.749861],[1.000000,0.000000,0.000000,0.000000],[0,0,-1,0],[9E+09,9E+09,9E+09,9E+09,9E+09,9E+09]];
    CONST robtarget T2223:=[[45.250631,33.503470,17.749861],[1.000000,0.000000,0.000000,0.000000],[0,0,-1,0],[9E+09,9E+09,9E+09,9E+09,9E+09,9E+09]];
    CONST robtarget T2224:=[[43.750625,33.963693,17.749861],[1.000000,0.000000,0.000000,0.000000],[0,0,-1,0],[9E+09,9E+09,9E+09,9E+09,9E+09,9E+09]];
    CONST robtarget T2225:=[[43.750625,76.133751,17.749861],[1.000000,0.000000,0.000000,0.000000],[0,0,-1,0],[9E+09,9E+09,9E+09,9E+09,9E+09,9E+09]];
    CONST robtarget T2226:=[[42.250619,74.508506,17.749861],[1.000000,0.000000,0.000000,0.000000],[0,0,-1,0],[9E+09,9E+09,9E+09,9E+09,9E+09,9E+09]];
    CONST robtarget T2227:=[[42.250619,34.588368,17.749861],[1.000000,0.000000,0.000000,0.000000],[0,0,-1,0],[9E+09,9E+09,9E+09,9E+09,9E+09,9E+09]];
    CONST robtarget T2228:=[[40.750613,35.306665,17.749861],[1.000000,0.000000,0.000000,0.000000],[0,0,-1,0],[9E+09,9E+09,9E+09,9E+09,9E+09,9E+09]];
    CONST robtarget T2229:=[[40.750613,72.416488,17.749861],[1.000000,0.000000,0.000000,0.000000],[0,0,-1,0],[9E+09,9E+09,9E+09,9E+09,9E+09,9E+09]];
    CONST robtarget T2230:=[[39.250607,70.257081,17.749861],[1.000000,0.000000,0.000000,0.000000],[0,0,-1,0],[9E+09,9E+09,9E+09,9E+09,9E+09,9E+09]];
    CONST robtarget T2231:=[[39.250607,36.287164,17.749861],[1.000000,0.000000,0.000000,0.000000],[0,0,-1,0],[9E+09,9E+09,9E+09,9E+09,9E+09,9E+09]];
    CONST robtarget T2232:=[[37.750601,37.525319,17.749861],[1.000000,0.000000,0.000000,0.000000],[0,0,-1,0],[9E+09,9E+09,9E+09,9E+09,9E+09,9E+09]];
    CONST robtarget T2233:=[[37.750601,71.929068,17.749861],[1.000000,0.000000,0.000000,0.000000],[0,0,-1,0],[9E+09,9E+09,9E+09,9E+09,9E+09,9E+09]];
    CONST robtarget T2234:=[[36.250595,70.038335,17.749861],[1.000000,0.000000,0.000000,0.000000],[0,0,-1,0],[9E+09,9E+09,9E+09,9E+09,9E+09,9E+09]];
    CONST robtarget T2235:=[[36.250595,39.278332,17.749861],[1.000000,0.000000,0.000000,0.000000],[0,0,-1,0],[9E+09,9E+09,9E+09,9E+09,9E+09,9E+09]];
    CONST robtarget T2236:=[[34.750589,41.729123,17.749861],[1.000000,0.000000,0.000000,0.000000],[0,0,-1,0],[9E+09,9E+09,9E+09,9E+09,9E+09,9E+09]];
    CONST robtarget T2237:=[[34.750589,66.382633,17.749861],[1.000000,0.000000,0.000000,0.000000],[0,0,-1,0],[9E+09,9E+09,9E+09,9E+09,9E+09,9E+09]];
    CONST robtarget T2238:=[[33.250583,61.052196,17.749861],[1.000000,0.000000,0.000000,0.000000],[0,0,-1,0],[9E+09,9E+09,9E+09,9E+09,9E+09,9E+09]];
    CONST robtarget T2239:=[[33.250583,48.947263,17.749861],[1.000000,0.000000,0.000000,0.000000],[0,0,-1,0],[9E+09,9E+09,9E+09,9E+09,9E+09,9E+09]];
    CONST robtarget T2240:=[[33.250515,51.514716,18.249871],[1.000000,0.000000,0.000000,0.000000],[0,0,-1,0],[9E+09,9E+09,9E+09,9E+09,9E+09,9E+09]];
    CONST robtarget T2241:=[[33.250515,59.637824,18.249871],[1.000000,0.000000,0.000000,0.000000],[0,0,-1,0],[9E+09,9E+09,9E+09,9E+09,9E+09,9E+09]];
    CONST robtarget T2242:=[[33.250515,51.514716,18.249871],[1.000000,0.000000,0.000000,0.000000],[0,0,-1,0],[9E+09,9E+09,9E+09,9E+09,9E+09,9E+09]];
    CONST robtarget T2243:=[[33.250515,59.637824,18.249871],[1.000000,0.000000,0.000000,0.000000],[0,0,-1,0],[9E+09,9E+09,9E+09,9E+09,9E+09,9E+09]];
    CONST robtarget T2244:=[[34.750521,65.865427,18.249871],[1.000000,0.000000,0.000000,0.000000],[0,0,-1,0],[9E+09,9E+09,9E+09,9E+09,9E+09,9E+09]];
    CONST robtarget T2245:=[[34.750521,42.533353,18.249871],[1.000000,0.000000,0.000000,0.000000],[0,0,-1,0],[9E+09,9E+09,9E+09,9E+09,9E+09,9E+09]];
    CONST robtarget T2246:=[[36.250527,39.694328,18.249871],[1.000000,0.000000,0.000000,0.000000],[0,0,-1,0],[9E+09,9E+09,9E+09,9E+09,9E+09,9E+09]];
    CONST robtarget T2247:=[[36.250527,69.741216,18.249871],[1.000000,0.000000,0.000000,0.000000],[0,0,-1,0],[9E+09,9E+09,9E+09,9E+09,9E+09,9E+09]];
    CONST robtarget T2248:=[[37.750533,71.942521,18.249871],[1.000000,0.000000,0.000000,0.000000],[0,0,-1,0],[9E+09,9E+09,9E+09,9E+09,9E+09,9E+09]];
    CONST robtarget T2249:=[[37.750533,37.920904,18.249871],[1.000000,0.000000,0.000000,0.000000],[0,0,-1,0],[9E+09,9E+09,9E+09,9E+09,9E+09,9E+09]];
    CONST robtarget T2250:=[[39.250539,36.538592,18.249871],[1.000000,0.000000,0.000000,0.000000],[0,0,-1,0],[9E+09,9E+09,9E+09,9E+09,9E+09,9E+09]];
    CONST robtarget T2251:=[[39.250539,70.189211,18.249871],[1.000000,0.000000,0.000000,0.000000],[0,0,-1,0],[9E+09,9E+09,9E+09,9E+09,9E+09,9E+09]];
    CONST robtarget T2252:=[[40.750545,72.282658,18.249871],[1.000000,0.000000,0.000000,0.000000],[0,0,-1,0],[9E+09,9E+09,9E+09,9E+09,9E+09,9E+09]];
    CONST robtarget T2253:=[[40.750545,35.558093,18.249871],[1.000000,0.000000,0.000000,0.000000],[0,0,-1,0],[9E+09,9E+09,9E+09,9E+09,9E+09,9E+09]];
    CONST robtarget T2254:=[[42.250551,34.808065,18.249871],[1.000000,0.000000,0.000000,0.000000],[0,0,-1,0],[9E+09,9E+09,9E+09,9E+09,9E+09,9E+09]];
    CONST robtarget T2255:=[[42.250551,74.394056,18.249871],[1.000000,0.000000,0.000000,0.000000],[0,0,-1,0],[9E+09,9E+09,9E+09,9E+09,9E+09,9E+09]];
    CONST robtarget T2256:=[[43.750557,76.094866,18.249871],[1.000000,0.000000,0.000000,0.000000],[0,0,-1,0],[9E+09,9E+09,9E+09,9E+09,9E+09,9E+09]];
    CONST robtarget T2257:=[[43.750557,34.183390,18.249871],[1.000000,0.000000,0.000000,0.000000],[0,0,-1,0],[9E+09,9E+09,9E+09,9E+09,9E+09,9E+09]];
    CONST robtarget T2258:=[[45.250563,33.700631,18.249871],[1.000000,0.000000,0.000000,0.000000],[0,0,-1,0],[9E+09,9E+09,9E+09,9E+09,9E+09,9E+09]];
    CONST robtarget T2259:=[[45.250563,77.189318,18.249871],[1.000000,0.000000,0.000000,0.000000],[0,0,-1,0],[9E+09,9E+09,9E+09,9E+09,9E+09,9E+09]];
    CONST robtarget T2260:=[[46.750569,77.923438,18.249871],[1.000000,0.000000,0.000000,0.000000],[0,0,-1,0],[9E+09,9E+09,9E+09,9E+09,9E+09,9E+09]];
    CONST robtarget T2261:=[[46.750569,33.323169,18.249871],[1.000000,0.000000,0.000000,0.000000],[0,0,-1,0],[9E+09,9E+09,9E+09,9E+09,9E+09,9E+09]];
    CONST robtarget T2262:=[[48.250575,33.017582,18.249871],[1.000000,0.000000,0.000000,0.000000],[0,0,-1,0],[9E+09,9E+09,9E+09,9E+09,9E+09,9E+09]];
    CONST robtarget T2263:=[[48.250575,78.446744,18.249871],[1.000000,0.000000,0.000000,0.000000],[0,0,-1,0],[9E+09,9E+09,9E+09,9E+09,9E+09,9E+09]];
    CONST robtarget T2264:=[[49.750581,78.885611,18.249871],[1.000000,0.000000,0.000000,0.000000],[0,0,-1,0],[9E+09,9E+09,9E+09,9E+09,9E+09,9E+09]];
    CONST robtarget T2265:=[[49.750581,32.801552,18.249871],[1.000000,0.000000,0.000000,0.000000],[0,0,-1,0],[9E+09,9E+09,9E+09,9E+09,9E+09,9E+09]];
    CONST robtarget T2266:=[[51.250587,32.631190,18.249871],[1.000000,0.000000,0.000000,0.000000],[0,0,-1,0],[9E+09,9E+09,9E+09,9E+09,9E+09,9E+09]];
    CONST robtarget T2267:=[[51.250587,79.205612,18.249871],[1.000000,0.000000,0.000000,0.000000],[0,0,-1,0],[9E+09,9E+09,9E+09,9E+09,9E+09,9E+09]];
    CONST robtarget T2268:=[[52.750593,79.492885,18.249871],[1.000000,0.000000,0.000000,0.000000],[0,0,-1,0],[9E+09,9E+09,9E+09,9E+09,9E+09,9E+09]];
    CONST robtarget T2269:=[[52.750593,32.515874,18.249871],[1.000000,0.000000,0.000000,0.000000],[0,0,-1,0],[9E+09,9E+09,9E+09,9E+09,9E+09,9E+09]];
    CONST robtarget T2270:=[[54.250599,32.486509,18.249871],[1.000000,0.000000,0.000000,0.000000],[0,0,-1,0],[9E+09,9E+09,9E+09,9E+09,9E+09,9E+09]];
    CONST robtarget T2271:=[[54.250599,79.819674,18.249871],[1.000000,0.000000,0.000000,0.000000],[0,0,-1,0],[9E+09,9E+09,9E+09,9E+09,9E+09,9E+09]];
    CONST robtarget T2272:=[[55.750605,79.819524,18.249871],[1.000000,0.000000,0.000000,0.000000],[0,0,-1,0],[9E+09,9E+09,9E+09,9E+09,9E+09,9E+09]];
    CONST robtarget T2273:=[[55.750605,32.486527,18.249871],[1.000000,0.000000,0.000000,0.000000],[0,0,-1,0],[9E+09,9E+09,9E+09,9E+09,9E+09,9E+09]];
    CONST robtarget T2274:=[[57.250611,32.515966,18.249871],[1.000000,0.000000,0.000000,0.000000],[0,0,-1,0],[9E+09,9E+09,9E+09,9E+09,9E+09,9E+09]];
    CONST robtarget T2275:=[[57.250611,79.492582,18.249871],[1.000000,0.000000,0.000000,0.000000],[0,0,-1,0],[9E+09,9E+09,9E+09,9E+09,9E+09,9E+09]];
    CONST robtarget T2276:=[[58.750617,79.205410,18.249871],[1.000000,0.000000,0.000000,0.000000],[0,0,-1,0],[9E+09,9E+09,9E+09,9E+09,9E+09,9E+09]];
    CONST robtarget T2277:=[[58.750617,32.631294,18.249871],[1.000000,0.000000,0.000000,0.000000],[0,0,-1,0],[9E+09,9E+09,9E+09,9E+09,9E+09,9E+09]];
    CONST robtarget T2278:=[[60.250623,32.801724,18.249871],[1.000000,0.000000,0.000000,0.000000],[0,0,-1,0],[9E+09,9E+09,9E+09,9E+09,9E+09,9E+09]];
    CONST robtarget T2279:=[[60.250623,78.885349,18.249871],[1.000000,0.000000,0.000000,0.000000],[0,0,-1,0],[9E+09,9E+09,9E+09,9E+09,9E+09,9E+09]];
    CONST robtarget T2280:=[[61.750629,78.446357,18.249871],[1.000000,0.000000,0.000000,0.000000],[0,0,-1,0],[9E+09,9E+09,9E+09,9E+09,9E+09,9E+09]];
    CONST robtarget T2281:=[[61.750629,33.017753,18.249871],[1.000000,0.000000,0.000000,0.000000],[0,0,-1,0],[9E+09,9E+09,9E+09,9E+09,9E+09,9E+09]];
    CONST robtarget T2282:=[[63.250635,33.323468,18.249871],[1.000000,0.000000,0.000000,0.000000],[0,0,-1,0],[9E+09,9E+09,9E+09,9E+09,9E+09,9E+09]];
    CONST robtarget T2283:=[[63.250635,77.922871,18.249871],[1.000000,0.000000,0.000000,0.000000],[0,0,-1,0],[9E+09,9E+09,9E+09,9E+09,9E+09,9E+09]];
    CONST robtarget T2284:=[[64.750641,77.188705,18.249871],[1.000000,0.000000,0.000000,0.000000],[0,0,-1,0],[9E+09,9E+09,9E+09,9E+09,9E+09,9E+09]];
    CONST robtarget T2285:=[[64.750641,33.700930,18.249871],[1.000000,0.000000,0.000000,0.000000],[0,0,-1,0],[9E+09,9E+09,9E+09,9E+09,9E+09,9E+09]];
    CONST robtarget T2286:=[[66.250647,34.183885,18.249871],[1.000000,0.000000,0.000000,0.000000],[0,0,-1,0],[9E+09,9E+09,9E+09,9E+09,9E+09,9E+09]];
    CONST robtarget T2287:=[[66.250647,76.093950,18.249871],[1.000000,0.000000,0.000000,0.000000],[0,0,-1,0],[9E+09,9E+09,9E+09,9E+09,9E+09,9E+09]];
    CONST robtarget T2288:=[[67.750653,74.392369,18.249871],[1.000000,0.000000,0.000000,0.000000],[0,0,-1,0],[9E+09,9E+09,9E+09,9E+09,9E+09,9E+09]];
    CONST robtarget T2289:=[[67.750653,34.808560,18.249871],[1.000000,0.000000,0.000000,0.000000],[0,0,-1,0],[9E+09,9E+09,9E+09,9E+09,9E+09,9E+09]];
    CONST robtarget T2290:=[[69.250659,35.558871,18.249871],[1.000000,0.000000,0.000000,0.000000],[0,0,-1,0],[9E+09,9E+09,9E+09,9E+09,9E+09,9E+09]];
    CONST robtarget T2291:=[[69.250659,72.280896,18.249871],[1.000000,0.000000,0.000000,0.000000],[0,0,-1,0],[9E+09,9E+09,9E+09,9E+09,9E+09,9E+09]];
    CONST robtarget T2292:=[[70.750665,70.187822,18.249871],[1.000000,0.000000,0.000000,0.000000],[0,0,-1,0],[9E+09,9E+09,9E+09,9E+09,9E+09,9E+09]];
    CONST robtarget T2293:=[[70.750665,36.539370,18.249871],[1.000000,0.000000,0.000000,0.000000],[0,0,-1,0],[9E+09,9E+09,9E+09,9E+09,9E+09,9E+09]];
    CONST robtarget T2294:=[[72.250671,37.922460,18.249871],[1.000000,0.000000,0.000000,0.000000],[0,0,-1,0],[9E+09,9E+09,9E+09,9E+09,9E+09,9E+09]];
    CONST robtarget T2295:=[[72.250671,71.942261,18.249871],[1.000000,0.000000,0.000000,0.000000],[0,0,-1,0],[9E+09,9E+09,9E+09,9E+09,9E+09,9E+09]];
    CONST robtarget T2296:=[[73.750677,69.739173,18.249871],[1.000000,0.000000,0.000000,0.000000],[0,0,-1,0],[9E+09,9E+09,9E+09,9E+09,9E+09,9E+09]];
    CONST robtarget T2297:=[[73.750677,39.695715,18.249871],[1.000000,0.000000,0.000000,0.000000],[0,0,-1,0],[9E+09,9E+09,9E+09,9E+09,9E+09,9E+09]];
    CONST robtarget T2298:=[[75.250683,42.536172,18.249871],[1.000000,0.000000,0.000000,0.000000],[0,0,-1,0],[9E+09,9E+09,9E+09,9E+09,9E+09,9E+09]];
    CONST robtarget T2299:=[[75.250683,65.881554,18.249871],[1.000000,0.000000,0.000000,0.000000],[0,0,-1,0],[9E+09,9E+09,9E+09,9E+09,9E+09,9E+09]];
    CONST robtarget T2300:=[[76.750689,59.668759,18.249871],[1.000000,0.000000,0.000000,0.000000],[0,0,-1,0],[9E+09,9E+09,9E+09,9E+09,9E+09,9E+09]];
    CONST robtarget T2301:=[[76.750689,51.520310,18.249871],[1.000000,0.000000,0.000000,0.000000],[0,0,-1,0],[9E+09,9E+09,9E+09,9E+09,9E+09,9E+09]];
    CONST robtarget T2302:=[[76.000619,51.020327,18.749881],[1.000000,0.000000,0.000000,0.000000],[0,0,-1,0],[9E+09,9E+09,9E+09,9E+09,9E+09,9E+09]];
    CONST robtarget T2303:=[[76.000619,61.950331,18.749881],[1.000000,0.000000,0.000000,0.000000],[0,0,-1,0],[9E+09,9E+09,9E+09,9E+09,9E+09,9E+09]];
    CONST robtarget T2304:=[[76.000619,51.020327,18.749881],[1.000000,0.000000,0.000000,0.000000],[0,0,-1,0],[9E+09,9E+09,9E+09,9E+09,9E+09,9E+09]];
    CONST robtarget T2305:=[[76.000619,61.950331,18.749881],[1.000000,0.000000,0.000000,0.000000],[0,0,-1,0],[9E+09,9E+09,9E+09,9E+09,9E+09,9E+09]];
    CONST robtarget T2306:=[[74.500613,67.596443,18.749881],[1.000000,0.000000,0.000000,0.000000],[0,0,-1,0],[9E+09,9E+09,9E+09,9E+09,9E+09,9E+09]];
    CONST robtarget T2307:=[[74.500613,41.612337,18.749881],[1.000000,0.000000,0.000000,0.000000],[0,0,-1,0],[9E+09,9E+09,9E+09,9E+09,9E+09,9E+09]];
    CONST robtarget T2308:=[[73.000607,39.237253,18.749881],[1.000000,0.000000,0.000000,0.000000],[0,0,-1,0],[9E+09,9E+09,9E+09,9E+09,9E+09,9E+09]];
    CONST robtarget T2309:=[[73.000607,70.835187,18.749881],[1.000000,0.000000,0.000000,0.000000],[0,0,-1,0],[9E+09,9E+09,9E+09,9E+09,9E+09,9E+09]];
    CONST robtarget T2310:=[[71.500601,72.207278,18.749881],[1.000000,0.000000,0.000000,0.000000],[0,0,-1,0],[9E+09,9E+09,9E+09,9E+09,9E+09,9E+09]];
    CONST robtarget T2311:=[[71.500601,37.337294,18.749881],[1.000000,0.000000,0.000000,0.000000],[0,0,-1,0],[9E+09,9E+09,9E+09,9E+09,9E+09,9E+09]];
    CONST robtarget T2312:=[[70.000595,36.300460,18.749881],[1.000000,0.000000,0.000000,0.000000],[0,0,-1,0],[9E+09,9E+09,9E+09,9E+09,9E+09,9E+09]];
    CONST robtarget T2313:=[[70.000595,71.042248,18.749881],[1.000000,0.000000,0.000000,0.000000],[0,0,-1,0],[9E+09,9E+09,9E+09,9E+09,9E+09,9E+09]];
    CONST robtarget T2314:=[[68.500589,73.221262,18.749881],[1.000000,0.000000,0.000000,0.000000],[0,0,-1,0],[9E+09,9E+09,9E+09,9E+09,9E+09,9E+09]];
    CONST robtarget T2315:=[[68.500589,35.340539,18.749881],[1.000000,0.000000,0.000000,0.000000],[0,0,-1,0],[9E+09,9E+09,9E+09,9E+09,9E+09,9E+09]];
    CONST robtarget T2316:=[[67.000583,34.715864,18.749881],[1.000000,0.000000,0.000000,0.000000],[0,0,-1,0],[9E+09,9E+09,9E+09,9E+09,9E+09,9E+09]];
    CONST robtarget T2317:=[[67.000583,75.186303,18.749881],[1.000000,0.000000,0.000000,0.000000],[0,0,-1,0],[9E+09,9E+09,9E+09,9E+09,9E+09,9E+09]];
    CONST robtarget T2318:=[[65.500577,76.632280,18.749881],[1.000000,0.000000,0.000000,0.000000],[0,0,-1,0],[9E+09,9E+09,9E+09,9E+09,9E+09,9E+09]];
    CONST robtarget T2319:=[[65.500577,34.106375,18.749881],[1.000000,0.000000,0.000000,0.000000],[0,0,-1,0],[9E+09,9E+09,9E+09,9E+09,9E+09,9E+09]];
    CONST robtarget T2320:=[[64.000571,33.720461,18.749881],[1.000000,0.000000,0.000000,0.000000],[0,0,-1,0],[9E+09,9E+09,9E+09,9E+09,9E+09,9E+09]];
    CONST robtarget T2321:=[[64.000571,77.542318,18.749881],[1.000000,0.000000,0.000000,0.000000],[0,0,-1,0],[9E+09,9E+09,9E+09,9E+09,9E+09,9E+09]];
    CONST robtarget T2322:=[[62.500565,78.190742,18.749881],[1.000000,0.000000,0.000000,0.000000],[0,0,-1,0],[9E+09,9E+09,9E+09,9E+09,9E+09,9E+09]];
    CONST robtarget T2323:=[[62.500565,33.342999,18.749881],[1.000000,0.000000,0.000000,0.000000],[0,0,-1,0],[9E+09,9E+09,9E+09,9E+09,9E+09,9E+09]];
    CONST robtarget T2324:=[[61.000559,33.110946,18.749881],[1.000000,0.000000,0.000000,0.000000],[0,0,-1,0],[9E+09,9E+09,9E+09,9E+09,9E+09,9E+09]];
    CONST robtarget T2325:=[[61.000559,78.707004,18.749881],[1.000000,0.000000,0.000000,0.000000],[0,0,-1,0],[9E+09,9E+09,9E+09,9E+09,9E+09,9E+09]];
    CONST robtarget T2326:=[[59.500553,79.048581,18.749881],[1.000000,0.000000,0.000000,0.000000],[0,0,-1,0],[9E+09,9E+09,9E+09,9E+09,9E+09,9E+09]];
    CONST robtarget T2327:=[[59.500553,32.896419,18.749881],[1.000000,0.000000,0.000000,0.000000],[0,0,-1,0],[9E+09,9E+09,9E+09,9E+09,9E+09,9E+09]];
    CONST robtarget T2328:=[[58.000547,32.766574,18.749881],[1.000000,0.000000,0.000000,0.000000],[0,0,-1,0],[9E+09,9E+09,9E+09,9E+09,9E+09,9E+09]];
    CONST robtarget T2329:=[[58.000547,79.331673,18.749881],[1.000000,0.000000,0.000000,0.000000],[0,0,-1,0],[9E+09,9E+09,9E+09,9E+09,9E+09,9E+09]];
    CONST robtarget T2330:=[[56.500541,79.669072,18.749881],[1.000000,0.000000,0.000000,0.000000],[0,0,-1,0],[9E+09,9E+09,9E+09,9E+09,9E+09,9E+09]];
    CONST robtarget T2331:=[[56.500541,32.672102,18.749881],[1.000000,0.000000,0.000000,0.000000],[0,0,-1,0],[9E+09,9E+09,9E+09,9E+09,9E+09,9E+09]];
    CONST robtarget T2332:=[[55.000535,32.633408,18.749881],[1.000000,0.000000,0.000000,0.000000],[0,0,-1,0],[9E+09,9E+09,9E+09,9E+09,9E+09,9E+09]];
    CONST robtarget T2333:=[[55.000535,79.916476,18.749881],[1.000000,0.000000,0.000000,0.000000],[0,0,-1,0],[9E+09,9E+09,9E+09,9E+09,9E+09,9E+09]];
    CONST robtarget T2334:=[[53.500529,79.669312,18.749881],[1.000000,0.000000,0.000000,0.000000],[0,0,-1,0],[9E+09,9E+09,9E+09,9E+09,9E+09,9E+09]];
    CONST robtarget T2335:=[[53.500529,32.672073,18.749881],[1.000000,0.000000,0.000000,0.000000],[0,0,-1,0],[9E+09,9E+09,9E+09,9E+09,9E+09,9E+09]];
    CONST robtarget T2336:=[[52.000523,32.766481,18.749881],[1.000000,0.000000,0.000000,0.000000],[0,0,-1,0],[9E+09,9E+09,9E+09,9E+09,9E+09,9E+09]];
    CONST robtarget T2337:=[[52.000523,79.331846,18.749881],[1.000000,0.000000,0.000000,0.000000],[0,0,-1,0],[9E+09,9E+09,9E+09,9E+09,9E+09,9E+09]];
    CONST robtarget T2338:=[[50.500517,79.048816,18.749881],[1.000000,0.000000,0.000000,0.000000],[0,0,-1,0],[9E+09,9E+09,9E+09,9E+09,9E+09,9E+09]];
    CONST robtarget T2339:=[[50.500517,32.896332,18.749881],[1.000000,0.000000,0.000000,0.000000],[0,0,-1,0],[9E+09,9E+09,9E+09,9E+09,9E+09,9E+09]];
    CONST robtarget T2340:=[[49.000511,33.110794,18.749881],[1.000000,0.000000,0.000000,0.000000],[0,0,-1,0],[9E+09,9E+09,9E+09,9E+09,9E+09,9E+09]];
    CONST robtarget T2341:=[[49.000511,78.707382,18.749881],[1.000000,0.000000,0.000000,0.000000],[0,0,-1,0],[9E+09,9E+09,9E+09,9E+09,9E+09,9E+09]];
    CONST robtarget T2342:=[[47.500505,78.191084,18.749881],[1.000000,0.000000,0.000000,0.000000],[0,0,-1,0],[9E+09,9E+09,9E+09,9E+09,9E+09,9E+09]];
    CONST robtarget T2343:=[[47.500505,33.342733,18.749881],[1.000000,0.000000,0.000000,0.000000],[0,0,-1,0],[9E+09,9E+09,9E+09,9E+09,9E+09,9E+09]];
    CONST robtarget T2344:=[[46.000499,33.720196,18.749881],[1.000000,0.000000,0.000000,0.000000],[0,0,-1,0],[9E+09,9E+09,9E+09,9E+09,9E+09,9E+09]];
    CONST robtarget T2345:=[[46.000499,77.542825,18.749881],[1.000000,0.000000,0.000000,0.000000],[0,0,-1,0],[9E+09,9E+09,9E+09,9E+09,9E+09,9E+09]];
    CONST robtarget T2346:=[[44.500493,76.633091,18.749881],[1.000000,0.000000,0.000000,0.000000],[0,0,-1,0],[9E+09,9E+09,9E+09,9E+09,9E+09,9E+09]];
    CONST robtarget T2347:=[[44.500493,34.105952,18.749881],[1.000000,0.000000,0.000000,0.000000],[0,0,-1,0],[9E+09,9E+09,9E+09,9E+09,9E+09,9E+09]];
    CONST robtarget T2348:=[[43.000487,34.715424,18.749881],[1.000000,0.000000,0.000000,0.000000],[0,0,-1,0],[9E+09,9E+09,9E+09,9E+09,9E+09,9E+09]];
    CONST robtarget T2349:=[[43.000487,75.187512,18.749881],[1.000000,0.000000,0.000000,0.000000],[0,0,-1,0],[9E+09,9E+09,9E+09,9E+09,9E+09,9E+09]];
    CONST robtarget T2350:=[[41.500481,73.222743,18.749881],[1.000000,0.000000,0.000000,0.000000],[0,0,-1,0],[9E+09,9E+09,9E+09,9E+09,9E+09,9E+09]];
    CONST robtarget T2351:=[[41.500481,35.340099,18.749881],[1.000000,0.000000,0.000000,0.000000],[0,0,-1,0],[9E+09,9E+09,9E+09,9E+09,9E+09,9E+09]];
    CONST robtarget T2352:=[[40.000475,36.299771,18.749881],[1.000000,0.000000,0.000000,0.000000],[0,0,-1,0],[9E+09,9E+09,9E+09,9E+09,9E+09,9E+09]];
    CONST robtarget T2353:=[[40.000475,71.043802,18.749881],[1.000000,0.000000,0.000000,0.000000],[0,0,-1,0],[9E+09,9E+09,9E+09,9E+09,9E+09,9E+09]];
    CONST robtarget T2354:=[[38.500469,72.207226,18.749881],[1.000000,0.000000,0.000000,0.000000],[0,0,-1,0],[9E+09,9E+09,9E+09,9E+09,9E+09,9E+09]];
    CONST robtarget T2355:=[[38.500469,37.335914,18.749881],[1.000000,0.000000,0.000000,0.000000],[0,0,-1,0],[9E+09,9E+09,9E+09,9E+09,9E+09,9E+09]];
    CONST robtarget T2356:=[[37.000463,39.236022,18.749881],[1.000000,0.000000,0.000000,0.000000],[0,0,-1,0],[9E+09,9E+09,9E+09,9E+09,9E+09,9E+09]];
    CONST robtarget T2357:=[[37.000463,70.836942,18.749881],[1.000000,0.000000,0.000000,0.000000],[0,0,-1,0],[9E+09,9E+09,9E+09,9E+09,9E+09,9E+09]];
    CONST robtarget T2358:=[[35.500457,67.591083,18.749881],[1.000000,0.000000,0.000000,0.000000],[0,0,-1,0],[9E+09,9E+09,9E+09,9E+09,9E+09,9E+09]];
    CONST robtarget T2359:=[[35.500457,41.609837,18.749881],[1.000000,0.000000,0.000000,0.000000],[0,0,-1,0],[9E+09,9E+09,9E+09,9E+09,9E+09,9E+09]];
    CONST robtarget T2360:=[[34.000451,51.016149,18.749881],[1.000000,0.000000,0.000000,0.000000],[0,0,-1,0],[9E+09,9E+09,9E+09,9E+09,9E+09,9E+09]];
    CONST robtarget T2361:=[[34.000451,61.900294,18.749881],[1.000000,0.000000,0.000000,0.000000],[0,0,-1,0],[9E+09,9E+09,9E+09,9E+09,9E+09,9E+09]];
    CONST robtarget T2362:=[[34.000383,54.227865,19.249891],[1.000000,0.000000,0.000000,0.000000],[0,0,-1,0],[9E+09,9E+09,9E+09,9E+09,9E+09,9E+09]];
    CONST robtarget T2363:=[[34.000383,60.409370,19.249891],[1.000000,0.000000,0.000000,0.000000],[0,0,-1,0],[9E+09,9E+09,9E+09,9E+09,9E+09,9E+09]];
    CONST robtarget T2364:=[[34.000383,54.227865,19.249891],[1.000000,0.000000,0.000000,0.000000],[0,0,-1,0],[9E+09,9E+09,9E+09,9E+09,9E+09,9E+09]];
    CONST robtarget T2365:=[[34.000383,60.409370,19.249891],[1.000000,0.000000,0.000000,0.000000],[0,0,-1,0],[9E+09,9E+09,9E+09,9E+09,9E+09,9E+09]];
    CONST robtarget T2366:=[[35.500389,66.864418,19.249891],[1.000000,0.000000,0.000000,0.000000],[0,0,-1,0],[9E+09,9E+09,9E+09,9E+09,9E+09,9E+09]];
    CONST robtarget T2367:=[[35.500389,42.462757,19.249891],[1.000000,0.000000,0.000000,0.000000],[0,0,-1,0],[9E+09,9E+09,9E+09,9E+09,9E+09,9E+09]];
    CONST robtarget T2368:=[[37.000395,39.652019,19.249891],[1.000000,0.000000,0.000000,0.000000],[0,0,-1,0],[9E+09,9E+09,9E+09,9E+09,9E+09,9E+09]];
    CONST robtarget T2369:=[[37.000395,70.600001,19.249891],[1.000000,0.000000,0.000000,0.000000],[0,0,-1,0],[9E+09,9E+09,9E+09,9E+09,9E+09,9E+09]];
    CONST robtarget T2370:=[[38.500401,72.309970,19.249891],[1.000000,0.000000,0.000000,0.000000],[0,0,-1,0],[9E+09,9E+09,9E+09,9E+09,9E+09,9E+09]];
    CONST robtarget T2371:=[[38.500401,37.731499,19.249891],[1.000000,0.000000,0.000000,0.000000],[0,0,-1,0],[9E+09,9E+09,9E+09,9E+09,9E+09,9E+09]];
    CONST robtarget T2372:=[[40.000407,36.559471,19.249891],[1.000000,0.000000,0.000000,0.000000],[0,0,-1,0],[9E+09,9E+09,9E+09,9E+09,9E+09,9E+09]];
    CONST robtarget T2373:=[[40.000407,70.796291,19.249891],[1.000000,0.000000,0.000000,0.000000],[0,0,-1,0],[9E+09,9E+09,9E+09,9E+09,9E+09,9E+09]];
    CONST robtarget T2374:=[[41.500413,72.956781,19.249891],[1.000000,0.000000,0.000000,0.000000],[0,0,-1,0],[9E+09,9E+09,9E+09,9E+09,9E+09,9E+09]];
    CONST robtarget T2375:=[[41.500413,35.570700,19.249891],[1.000000,0.000000,0.000000,0.000000],[0,0,-1,0],[9E+09,9E+09,9E+09,9E+09,9E+09,9E+09]];
    CONST robtarget T2376:=[[43.000419,34.935121,19.249891],[1.000000,0.000000,0.000000,0.000000],[0,0,-1,0],[9E+09,9E+09,9E+09,9E+09,9E+09,9E+09]];
    CONST robtarget T2377:=[[43.000419,75.046032,19.249891],[1.000000,0.000000,0.000000,0.000000],[0,0,-1,0],[9E+09,9E+09,9E+09,9E+09,9E+09,9E+09]];
    CONST robtarget T2378:=[[44.500425,76.559966,19.249891],[1.000000,0.000000,0.000000,0.000000],[0,0,-1,0],[9E+09,9E+09,9E+09,9E+09,9E+09,9E+09]];
    CONST robtarget T2379:=[[44.500425,34.331478,19.249891],[1.000000,0.000000,0.000000,0.000000],[0,0,-1,0],[9E+09,9E+09,9E+09,9E+09,9E+09,9E+09]];
    CONST robtarget T2380:=[[46.000431,33.928492,19.249891],[1.000000,0.000000,0.000000,0.000000],[0,0,-1,0],[9E+09,9E+09,9E+09,9E+09,9E+09,9E+09]];
    CONST robtarget T2381:=[[46.000431,77.517285,19.249891],[1.000000,0.000000,0.000000,0.000000],[0,0,-1,0],[9E+09,9E+09,9E+09,9E+09,9E+09,9E+09]];
    CONST robtarget T2382:=[[47.500437,78.186552,19.249891],[1.000000,0.000000,0.000000,0.000000],[0,0,-1,0],[9E+09,9E+09,9E+09,9E+09,9E+09,9E+09]];
    CONST robtarget T2383:=[[47.500437,33.551029,19.249891],[1.000000,0.000000,0.000000,0.000000],[0,0,-1,0],[9E+09,9E+09,9E+09,9E+09,9E+09,9E+09]];
    CONST robtarget T2384:=[[49.000443,33.312020,19.249891],[1.000000,0.000000,0.000000,0.000000],[0,0,-1,0],[9E+09,9E+09,9E+09,9E+09,9E+09,9E+09]];
    CONST robtarget T2385:=[[49.000443,78.694258,19.249891],[1.000000,0.000000,0.000000,0.000000],[0,0,-1,0],[9E+09,9E+09,9E+09,9E+09,9E+09,9E+09]];
    CONST robtarget T2386:=[[50.500449,79.043192,19.249891],[1.000000,0.000000,0.000000,0.000000],[0,0,-1,0],[9E+09,9E+09,9E+09,9E+09,9E+09,9E+09]];
    CONST robtarget T2387:=[[50.500449,33.098429,19.249891],[1.000000,0.000000,0.000000,0.000000],[0,0,-1,0],[9E+09,9E+09,9E+09,9E+09,9E+09,9E+09]];
    CONST robtarget T2388:=[[52.000455,32.967451,19.249891],[1.000000,0.000000,0.000000,0.000000],[0,0,-1,0],[9E+09,9E+09,9E+09,9E+09,9E+09,9E+09]];
    CONST robtarget T2389:=[[52.000455,79.328460,19.249891],[1.000000,0.000000,0.000000,0.000000],[0,0,-1,0],[9E+09,9E+09,9E+09,9E+09,9E+09,9E+09]];
    CONST robtarget T2390:=[[53.500461,79.656638,19.249891],[1.000000,0.000000,0.000000,0.000000],[0,0,-1,0],[9E+09,9E+09,9E+09,9E+09,9E+09,9E+09]];
    CONST robtarget T2391:=[[53.500461,32.871575,19.249891],[1.000000,0.000000,0.000000,0.000000],[0,0,-1,0],[9E+09,9E+09,9E+09,9E+09,9E+09,9E+09]];
    CONST robtarget T2392:=[[55.000467,32.838376,19.249891],[1.000000,0.000000,0.000000,0.000000],[0,0,-1,0],[9E+09,9E+09,9E+09,9E+09,9E+09,9E+09]];
    CONST robtarget T2393:=[[55.000467,79.901605,19.249891],[1.000000,0.000000,0.000000,0.000000],[0,0,-1,0],[9E+09,9E+09,9E+09,9E+09,9E+09,9E+09]];
    CONST robtarget T2394:=[[56.500473,79.656430,19.249891],[1.000000,0.000000,0.000000,0.000000],[0,0,-1,0],[9E+09,9E+09,9E+09,9E+09,9E+09,9E+09]];
    CONST robtarget T2395:=[[56.500473,32.871601,19.249891],[1.000000,0.000000,0.000000,0.000000],[0,0,-1,0],[9E+09,9E+09,9E+09,9E+09,9E+09,9E+09]];
    CONST robtarget T2396:=[[58.000479,32.967532,19.249891],[1.000000,0.000000,0.000000,0.000000],[0,0,-1,0],[9E+09,9E+09,9E+09,9E+09,9E+09,9E+09]];
    CONST robtarget T2397:=[[58.000479,79.328311,19.249891],[1.000000,0.000000,0.000000,0.000000],[0,0,-1,0],[9E+09,9E+09,9E+09,9E+09,9E+09,9E+09]];
    CONST robtarget T2398:=[[59.500485,79.042987,19.249891],[1.000000,0.000000,0.000000,0.000000],[0,0,-1,0],[9E+09,9E+09,9E+09,9E+09,9E+09,9E+09]];
    CONST robtarget T2399:=[[59.500485,33.098559,19.249891],[1.000000,0.000000,0.000000,0.000000],[0,0,-1,0],[9E+09,9E+09,9E+09,9E+09,9E+09,9E+09]];
    CONST robtarget T2400:=[[61.000491,33.312153,19.249891],[1.000000,0.000000,0.000000,0.000000],[0,0,-1,0],[9E+09,9E+09,9E+09,9E+09,9E+09,9E+09]];
    CONST robtarget T2401:=[[61.000491,78.693931,19.249891],[1.000000,0.000000,0.000000,0.000000],[0,0,-1,0],[9E+09,9E+09,9E+09,9E+09,9E+09,9E+09]];
    CONST robtarget T2402:=[[62.500497,78.186255,19.249891],[1.000000,0.000000,0.000000,0.000000],[0,0,-1,0],[9E+09,9E+09,9E+09,9E+09,9E+09,9E+09]];
    CONST robtarget T2403:=[[62.500497,33.551261,19.249891],[1.000000,0.000000,0.000000,0.000000],[0,0,-1,0],[9E+09,9E+09,9E+09,9E+09,9E+09,9E+09]];
    CONST robtarget T2404:=[[64.000503,33.928723,19.249891],[1.000000,0.000000,0.000000,0.000000],[0,0,-1,0],[9E+09,9E+09,9E+09,9E+09,9E+09,9E+09]];
    CONST robtarget T2405:=[[64.000503,77.516830,19.249891],[1.000000,0.000000,0.000000,0.000000],[0,0,-1,0],[9E+09,9E+09,9E+09,9E+09,9E+09,9E+09]];
    CONST robtarget T2406:=[[65.500509,76.559249,19.249891],[1.000000,0.000000,0.000000,0.000000],[0,0,-1,0],[9E+09,9E+09,9E+09,9E+09,9E+09,9E+09]];
    CONST robtarget T2407:=[[65.500509,34.331846,19.249891],[1.000000,0.000000,0.000000,0.000000],[0,0,-1,0],[9E+09,9E+09,9E+09,9E+09,9E+09,9E+09]];
    CONST robtarget T2408:=[[67.000515,34.935504,19.249891],[1.000000,0.000000,0.000000,0.000000],[0,0,-1,0],[9E+09,9E+09,9E+09,9E+09,9E+09,9E+09]];
    CONST robtarget T2409:=[[67.000515,75.044967,19.249891],[1.000000,0.000000,0.000000,0.000000],[0,0,-1,0],[9E+09,9E+09,9E+09,9E+09,9E+09,9E+09]];
    CONST robtarget T2410:=[[68.500521,72.955453,19.249891],[1.000000,0.000000,0.000000,0.000000],[0,0,-1,0],[9E+09,9E+09,9E+09,9E+09,9E+09,9E+09]];
    CONST robtarget T2411:=[[68.500521,35.571301,19.249891],[1.000000,0.000000,0.000000,0.000000],[0,0,-1,0],[9E+09,9E+09,9E+09,9E+09,9E+09,9E+09]];
    CONST robtarget T2412:=[[70.000527,36.560108,19.249891],[1.000000,0.000000,0.000000,0.000000],[0,0,-1,0],[9E+09,9E+09,9E+09,9E+09,9E+09,9E+09]];
    CONST robtarget T2413:=[[70.000527,70.795645,19.249891],[1.000000,0.000000,0.000000,0.000000],[0,0,-1,0],[9E+09,9E+09,9E+09,9E+09,9E+09,9E+09]];
    CONST robtarget T2414:=[[71.500533,72.309533,19.249891],[1.000000,0.000000,0.000000,0.000000],[0,0,-1,0],[9E+09,9E+09,9E+09,9E+09,9E+09,9E+09]];
    CONST robtarget T2415:=[[71.500533,37.732703,19.249891],[1.000000,0.000000,0.000000,0.000000],[0,0,-1,0],[9E+09,9E+09,9E+09,9E+09,9E+09,9E+09]];
    CONST robtarget T2416:=[[73.000539,39.653092,19.249891],[1.000000,0.000000,0.000000,0.000000],[0,0,-1,0],[9E+09,9E+09,9E+09,9E+09,9E+09,9E+09]];
    CONST robtarget T2417:=[[73.000539,70.598435,19.249891],[1.000000,0.000000,0.000000,0.000000],[0,0,-1,0],[9E+09,9E+09,9E+09,9E+09,9E+09,9E+09]];
    CONST robtarget T2418:=[[74.500545,66.879010,19.249891],[1.000000,0.000000,0.000000,0.000000],[0,0,-1,0],[9E+09,9E+09,9E+09,9E+09,9E+09,9E+09]];
    CONST robtarget T2419:=[[74.500545,42.464937,19.249891],[1.000000,0.000000,0.000000,0.000000],[0,0,-1,0],[9E+09,9E+09,9E+09,9E+09,9E+09,9E+09]];
    CONST robtarget T2420:=[[76.000551,54.234659,19.249891],[1.000000,0.000000,0.000000,0.000000],[0,0,-1,0],[9E+09,9E+09,9E+09,9E+09,9E+09,9E+09]];
    CONST robtarget T2421:=[[76.000551,60.444189,19.249891],[1.000000,0.000000,0.000000,0.000000],[0,0,-1,0],[9E+09,9E+09,9E+09,9E+09,9E+09,9E+09]];
    CONST robtarget T2422:=[[75.249803,53.625265,19.749901],[1.000000,0.000000,0.000000,0.000000],[0,0,-1,0],[9E+09,9E+09,9E+09,9E+09,9E+09,9E+09]];
    CONST robtarget T2423:=[[75.249803,62.924155,19.749901],[1.000000,0.000000,0.000000,0.000000],[0,0,-1,0],[9E+09,9E+09,9E+09,9E+09,9E+09,9E+09]];
    CONST robtarget T2424:=[[75.249803,53.625265,19.749901],[1.000000,0.000000,0.000000,0.000000],[0,0,-1,0],[9E+09,9E+09,9E+09,9E+09,9E+09,9E+09]];
    CONST robtarget T2425:=[[75.249803,62.924155,19.749901],[1.000000,0.000000,0.000000,0.000000],[0,0,-1,0],[9E+09,9E+09,9E+09,9E+09,9E+09,9E+09]];
    CONST robtarget T2426:=[[73.749797,68.517332,19.749901],[1.000000,0.000000,0.000000,0.000000],[0,0,-1,0],[9E+09,9E+09,9E+09,9E+09,9E+09,9E+09]];
    CONST robtarget T2427:=[[73.749797,41.539497,19.749901],[1.000000,0.000000,0.000000,0.000000],[0,0,-1,0],[9E+09,9E+09,9E+09,9E+09,9E+09,9E+09]];
    CONST robtarget T2428:=[[72.249791,39.107802,19.749901],[1.000000,0.000000,0.000000,0.000000],[0,0,-1,0],[9E+09,9E+09,9E+09,9E+09,9E+09,9E+09]];
    CONST robtarget T2429:=[[72.249791,71.632913,19.749901],[1.000000,0.000000,0.000000,0.000000],[0,0,-1,0],[9E+09,9E+09,9E+09,9E+09,9E+09,9E+09]];
    CONST robtarget T2430:=[[70.749785,72.337268,19.749901],[1.000000,0.000000,0.000000,0.000000],[0,0,-1,0],[9E+09,9E+09,9E+09,9E+09,9E+09,9E+09]];
    CONST robtarget T2431:=[[70.749785,37.353004,19.749901],[1.000000,0.000000,0.000000,0.000000],[0,0,-1,0],[9E+09,9E+09,9E+09,9E+09,9E+09,9E+09]];
    CONST robtarget T2432:=[[69.249779,36.313091,19.749901],[1.000000,0.000000,0.000000,0.000000],[0,0,-1,0],[9E+09,9E+09,9E+09,9E+09,9E+09,9E+09]];
    CONST robtarget T2433:=[[69.249779,71.565066,19.749901],[1.000000,0.000000,0.000000,0.000000],[0,0,-1,0],[9E+09,9E+09,9E+09,9E+09,9E+09,9E+09]];
    CONST robtarget T2434:=[[67.749773,73.722568,19.749901],[1.000000,0.000000,0.000000,0.000000],[0,0,-1,0],[9E+09,9E+09,9E+09,9E+09,9E+09,9E+09]];
    CONST robtarget T2435:=[[67.749773,35.467201,19.749901],[1.000000,0.000000,0.000000,0.000000],[0,0,-1,0],[9E+09,9E+09,9E+09,9E+09,9E+09,9E+09]];
    CONST robtarget T2436:=[[66.249767,34.857702,19.749901],[1.000000,0.000000,0.000000,0.000000],[0,0,-1,0],[9E+09,9E+09,9E+09,9E+09,9E+09,9E+09]];
    CONST robtarget T2437:=[[66.249767,75.720860,19.749901],[1.000000,0.000000,0.000000,0.000000],[0,0,-1,0],[9E+09,9E+09,9E+09,9E+09,9E+09,9E+09]];
    CONST robtarget T2438:=[[64.749761,77.012424,19.749901],[1.000000,0.000000,0.000000,0.000000],[0,0,-1,0],[9E+09,9E+09,9E+09,9E+09,9E+09,9E+09]];
    CONST robtarget T2439:=[[64.749761,34.332216,19.749901],[1.000000,0.000000,0.000000,0.000000],[0,0,-1,0],[9E+09,9E+09,9E+09,9E+09,9E+09,9E+09]];
    CONST robtarget T2440:=[[63.249755,33.948083,19.749901],[1.000000,0.000000,0.000000,0.000000],[0,0,-1,0],[9E+09,9E+09,9E+09,9E+09,9E+09,9E+09]];
    CONST robtarget T2441:=[[63.249755,77.796569,19.749901],[1.000000,0.000000,0.000000,0.000000],[0,0,-1,0],[9E+09,9E+09,9E+09,9E+09,9E+09,9E+09]];
    CONST robtarget T2442:=[[61.749749,78.409321,19.749901],[1.000000,0.000000,0.000000,0.000000],[0,0,-1,0],[9E+09,9E+09,9E+09,9E+09,9E+09,9E+09]];
    CONST robtarget T2443:=[[61.749749,33.621277,19.749901],[1.000000,0.000000,0.000000,0.000000],[0,0,-1,0],[9E+09,9E+09,9E+09,9E+09,9E+09,9E+09]];
    CONST robtarget T2444:=[[60.249743,33.406538,19.749901],[1.000000,0.000000,0.000000,0.000000],[0,0,-1,0],[9E+09,9E+09,9E+09,9E+09,9E+09,9E+09]];
    CONST robtarget T2445:=[[60.249743,78.868720,19.749901],[1.000000,0.000000,0.000000,0.000000],[0,0,-1,0],[9E+09,9E+09,9E+09,9E+09,9E+09,9E+09]];
    CONST robtarget T2446:=[[58.749737,79.195440,19.749901],[1.000000,0.000000,0.000000,0.000000],[0,0,-1,0],[9E+09,9E+09,9E+09,9E+09,9E+09,9E+09]];
    CONST robtarget T2447:=[[58.749737,33.232908,19.749901],[1.000000,0.000000,0.000000,0.000000],[0,0,-1,0],[9E+09,9E+09,9E+09,9E+09,9E+09,9E+09]];
    CONST robtarget T2448:=[[57.249731,33.102752,19.749901],[1.000000,0.000000,0.000000,0.000000],[0,0,-1,0],[9E+09,9E+09,9E+09,9E+09,9E+09,9E+09]];
    CONST robtarget T2449:=[[57.249731,79.465749,19.749901],[1.000000,0.000000,0.000000,0.000000],[0,0,-1,0],[9E+09,9E+09,9E+09,9E+09,9E+09,9E+09]];
    CONST robtarget T2450:=[[55.749725,79.784644,19.749901],[1.000000,0.000000,0.000000,0.000000],[0,0,-1,0],[9E+09,9E+09,9E+09,9E+09,9E+09,9E+09]];
    CONST robtarget T2451:=[[55.749725,33.049969,19.749901],[1.000000,0.000000,0.000000,0.000000],[0,0,-1,0],[9E+09,9E+09,9E+09,9E+09,9E+09,9E+09]];
    CONST robtarget T2452:=[[54.249719,33.049985,19.749901],[1.000000,0.000000,0.000000,0.000000],[0,0,-1,0],[9E+09,9E+09,9E+09,9E+09,9E+09,9E+09]];
    CONST robtarget T2453:=[[54.249719,79.784572,19.749901],[1.000000,0.000000,0.000000,0.000000],[0,0,-1,0],[9E+09,9E+09,9E+09,9E+09,9E+09,9E+09]];
    CONST robtarget T2454:=[[52.749713,79.465587,19.749901],[1.000000,0.000000,0.000000,0.000000],[0,0,-1,0],[9E+09,9E+09,9E+09,9E+09,9E+09,9E+09]];
    CONST robtarget T2455:=[[52.749713,33.102802,19.749901],[1.000000,0.000000,0.000000,0.000000],[0,0,-1,0],[9E+09,9E+09,9E+09,9E+09,9E+09,9E+09]];
    CONST robtarget T2456:=[[51.249707,33.232955,19.749901],[1.000000,0.000000,0.000000,0.000000],[0,0,-1,0],[9E+09,9E+09,9E+09,9E+09,9E+09,9E+09]];
    CONST robtarget T2457:=[[51.249707,79.195340,19.749901],[1.000000,0.000000,0.000000,0.000000],[0,0,-1,0],[9E+09,9E+09,9E+09,9E+09,9E+09,9E+09]];
    CONST robtarget T2458:=[[49.749701,78.868585,19.749901],[1.000000,0.000000,0.000000,0.000000],[0,0,-1,0],[9E+09,9E+09,9E+09,9E+09,9E+09,9E+09]];
    CONST robtarget T2459:=[[49.749701,33.406618,19.749901],[1.000000,0.000000,0.000000,0.000000],[0,0,-1,0],[9E+09,9E+09,9E+09,9E+09,9E+09,9E+09]];
    CONST robtarget T2460:=[[48.249695,33.621359,19.749901],[1.000000,0.000000,0.000000,0.000000],[0,0,-1,0],[9E+09,9E+09,9E+09,9E+09,9E+09,9E+09]];
    CONST robtarget T2461:=[[48.249695,78.409097,19.749901],[1.000000,0.000000,0.000000,0.000000],[0,0,-1,0],[9E+09,9E+09,9E+09,9E+09,9E+09,9E+09]];
    CONST robtarget T2462:=[[46.749689,77.796274,19.749901],[1.000000,0.000000,0.000000,0.000000],[0,0,-1,0],[9E+09,9E+09,9E+09,9E+09,9E+09,9E+09]];
    CONST robtarget T2463:=[[46.749689,33.948227,19.749901],[1.000000,0.000000,0.000000,0.000000],[0,0,-1,0],[9E+09,9E+09,9E+09,9E+09,9E+09,9E+09]];
    CONST robtarget T2464:=[[45.249683,34.332363,19.749901],[1.000000,0.000000,0.000000,0.000000],[0,0,-1,0],[9E+09,9E+09,9E+09,9E+09,9E+09,9E+09]];
    CONST robtarget T2465:=[[45.249683,77.011950,19.749901],[1.000000,0.000000,0.000000,0.000000],[0,0,-1,0],[9E+09,9E+09,9E+09,9E+09,9E+09,9E+09]];
    CONST robtarget T2466:=[[43.749677,75.720201,19.749901],[1.000000,0.000000,0.000000,0.000000],[0,0,-1,0],[9E+09,9E+09,9E+09,9E+09,9E+09,9E+09]];
    CONST robtarget T2467:=[[43.749677,34.857931,19.749901],[1.000000,0.000000,0.000000,0.000000],[0,0,-1,0],[9E+09,9E+09,9E+09,9E+09,9E+09,9E+09]];
    CONST robtarget T2468:=[[42.249671,35.467438,19.749901],[1.000000,0.000000,0.000000,0.000000],[0,0,-1,0],[9E+09,9E+09,9E+09,9E+09,9E+09,9E+09]];
    CONST robtarget T2469:=[[42.249671,73.721755,19.749901],[1.000000,0.000000,0.000000,0.000000],[0,0,-1,0],[9E+09,9E+09,9E+09,9E+09,9E+09,9E+09]];
    CONST robtarget T2470:=[[40.749665,71.564244,19.749901],[1.000000,0.000000,0.000000,0.000000],[0,0,-1,0],[9E+09,9E+09,9E+09,9E+09,9E+09,9E+09]];
    CONST robtarget T2471:=[[40.749665,36.313486,19.749901],[1.000000,0.000000,0.000000,0.000000],[0,0,-1,0],[9E+09,9E+09,9E+09,9E+09,9E+09,9E+09]];
    CONST robtarget T2472:=[[39.249659,37.353399,19.749901],[1.000000,0.000000,0.000000,0.000000],[0,0,-1,0],[9E+09,9E+09,9E+09,9E+09,9E+09,9E+09]];
    CONST robtarget T2473:=[[39.249659,72.337778,19.749901],[1.000000,0.000000,0.000000,0.000000],[0,0,-1,0],[9E+09,9E+09,9E+09,9E+09,9E+09,9E+09]];
    CONST robtarget T2474:=[[37.749653,71.631965,19.749901],[1.000000,0.000000,0.000000,0.000000],[0,0,-1,0],[9E+09,9E+09,9E+09,9E+09,9E+09,9E+09]];
    CONST robtarget T2475:=[[37.749653,39.108546,19.749901],[1.000000,0.000000,0.000000,0.000000],[0,0,-1,0],[9E+09,9E+09,9E+09,9E+09,9E+09,9E+09]];
    CONST robtarget T2476:=[[36.249647,41.540845,19.749901],[1.000000,0.000000,0.000000,0.000000],[0,0,-1,0],[9E+09,9E+09,9E+09,9E+09,9E+09,9E+09]];
    CONST robtarget T2477:=[[36.249647,68.510724,19.749901],[1.000000,0.000000,0.000000,0.000000],[0,0,-1,0],[9E+09,9E+09,9E+09,9E+09,9E+09,9E+09]];
    CONST robtarget T2478:=[[34.749641,62.859839,19.749901],[1.000000,0.000000,0.000000,0.000000],[0,0,-1,0],[9E+09,9E+09,9E+09,9E+09,9E+09,9E+09]];
    CONST robtarget T2479:=[[34.749641,53.628354,19.749901],[1.000000,0.000000,0.000000,0.000000],[0,0,-1,0],[9E+09,9E+09,9E+09,9E+09,9E+09,9E+09]];
    CONST robtarget T2480:=[[35.499029,53.932751,20.249911],[1.000000,0.000000,0.000000,0.000000],[0,0,-1,0],[9E+09,9E+09,9E+09,9E+09,9E+09,9E+09]];
    CONST robtarget T2481:=[[35.499029,64.959018,20.249911],[1.000000,0.000000,0.000000,0.000000],[0,0,-1,0],[9E+09,9E+09,9E+09,9E+09,9E+09,9E+09]];
    CONST robtarget T2482:=[[35.499029,53.932751,20.249911],[1.000000,0.000000,0.000000,0.000000],[0,0,-1,0],[9E+09,9E+09,9E+09,9E+09,9E+09,9E+09]];
    CONST robtarget T2483:=[[35.499029,64.959018,20.249911],[1.000000,0.000000,0.000000,0.000000],[0,0,-1,0],[9E+09,9E+09,9E+09,9E+09,9E+09,9E+09]];
    CONST robtarget T2484:=[[36.999035,69.842386,20.249911],[1.000000,0.000000,0.000000,0.000000],[0,0,-1,0],[9E+09,9E+09,9E+09,9E+09,9E+09,9E+09]];
    CONST robtarget T2485:=[[36.999035,40.728652,20.249911],[1.000000,0.000000,0.000000,0.000000],[0,0,-1,0],[9E+09,9E+09,9E+09,9E+09,9E+09,9E+09]];
    CONST robtarget T2486:=[[38.499041,38.524271,20.249911],[1.000000,0.000000,0.000000,0.000000],[0,0,-1,0],[9E+09,9E+09,9E+09,9E+09,9E+09,9E+09]];
    CONST robtarget T2487:=[[38.499041,72.380374,20.249911],[1.000000,0.000000,0.000000,0.000000],[0,0,-1,0],[9E+09,9E+09,9E+09,9E+09,9E+09,9E+09]];
    CONST robtarget T2488:=[[39.999047,70.367548,20.249911],[1.000000,0.000000,0.000000,0.000000],[0,0,-1,0],[9E+09,9E+09,9E+09,9E+09,9E+09,9E+09]];
    CONST robtarget T2489:=[[39.999047,37.107324,20.249911],[1.000000,0.000000,0.000000,0.000000],[0,0,-1,0],[9E+09,9E+09,9E+09,9E+09,9E+09,9E+09]];
    CONST robtarget T2490:=[[41.499053,36.074357,20.249911],[1.000000,0.000000,0.000000,0.000000],[0,0,-1,0],[9E+09,9E+09,9E+09,9E+09,9E+09,9E+09]];
    CONST robtarget T2491:=[[41.499053,72.335647,20.249911],[1.000000,0.000000,0.000000,0.000000],[0,0,-1,0],[9E+09,9E+09,9E+09,9E+09,9E+09,9E+09]];
    CONST robtarget T2492:=[[42.999059,74.593946,20.249911],[1.000000,0.000000,0.000000,0.000000],[0,0,-1,0],[9E+09,9E+09,9E+09,9E+09,9E+09,9E+09]];
    CONST robtarget T2493:=[[42.999059,35.384332,20.249911],[1.000000,0.000000,0.000000,0.000000],[0,0,-1,0],[9E+09,9E+09,9E+09,9E+09,9E+09,9E+09]];
    CONST robtarget T2494:=[[44.499065,34.783021,20.249911],[1.000000,0.000000,0.000000,0.000000],[0,0,-1,0],[9E+09,9E+09,9E+09,9E+09,9E+09,9E+09]];
    CONST robtarget T2495:=[[44.499065,76.287195,20.249911],[1.000000,0.000000,0.000000,0.000000],[0,0,-1,0],[9E+09,9E+09,9E+09,9E+09,9E+09,9E+09]];
    CONST robtarget T2496:=[[45.999071,77.323280,20.249911],[1.000000,0.000000,0.000000,0.000000],[0,0,-1,0],[9E+09,9E+09,9E+09,9E+09,9E+09,9E+09]];
    CONST robtarget T2497:=[[45.999071,34.350358,20.249911],[1.000000,0.000000,0.000000,0.000000],[0,0,-1,0],[9E+09,9E+09,9E+09,9E+09,9E+09,9E+09]];
    CONST robtarget T2498:=[[47.499077,33.967929,20.249911],[1.000000,0.000000,0.000000,0.000000],[0,0,-1,0],[9E+09,9E+09,9E+09,9E+09,9E+09,9E+09]];
    CONST robtarget T2499:=[[47.499077,78.045890,20.249911],[1.000000,0.000000,0.000000,0.000000],[0,0,-1,0],[9E+09,9E+09,9E+09,9E+09,9E+09,9E+09]];
    CONST robtarget T2500:=[[48.999083,78.607188,20.249911],[1.000000,0.000000,0.000000,0.000000],[0,0,-1,0],[9E+09,9E+09,9E+09,9E+09,9E+09,9E+09]];
    CONST robtarget T2501:=[[48.999083,33.714788,20.249911],[1.000000,0.000000,0.000000,0.000000],[0,0,-1,0],[9E+09,9E+09,9E+09,9E+09,9E+09,9E+09]];
    CONST robtarget T2502:=[[50.499089,33.503241,20.249911],[1.000000,0.000000,0.000000,0.000000],[0,0,-1,0],[9E+09,9E+09,9E+09,9E+09,9E+09,9E+09]];
    CONST robtarget T2503:=[[50.499089,78.997617,20.249911],[1.000000,0.000000,0.000000,0.000000],[0,0,-1,0],[9E+09,9E+09,9E+09,9E+09,9E+09,9E+09]];
    CONST robtarget T2504:=[[51.999095,79.321478,20.249911],[1.000000,0.000000,0.000000,0.000000],[0,0,-1,0],[9E+09,9E+09,9E+09,9E+09,9E+09,9E+09]];
    CONST robtarget T2505:=[[51.999095,33.369497,20.249911],[1.000000,0.000000,0.000000,0.000000],[0,0,-1,0],[9E+09,9E+09,9E+09,9E+09,9E+09,9E+09]];
    CONST robtarget T2506:=[[53.499101,33.270614,20.249911],[1.000000,0.000000,0.000000,0.000000],[0,0,-1,0],[9E+09,9E+09,9E+09,9E+09,9E+09,9E+09]];
    CONST robtarget T2507:=[[53.499101,79.631006,20.249911],[1.000000,0.000000,0.000000,0.000000],[0,0,-1,0],[9E+09,9E+09,9E+09,9E+09,9E+09,9E+09]];
    CONST robtarget T2508:=[[54.999107,79.871772,20.249911],[1.000000,0.000000,0.000000,0.000000],[0,0,-1,0],[9E+09,9E+09,9E+09,9E+09,9E+09,9E+09]];
    CONST robtarget T2509:=[[54.999107,33.248315,20.249911],[1.000000,0.000000,0.000000,0.000000],[0,0,-1,0],[9E+09,9E+09,9E+09,9E+09,9E+09,9E+09]];
    CONST robtarget T2510:=[[56.499113,33.270563,20.249911],[1.000000,0.000000,0.000000,0.000000],[0,0,-1,0],[9E+09,9E+09,9E+09,9E+09,9E+09,9E+09]];
    CONST robtarget T2511:=[[56.499113,79.631429,20.249911],[1.000000,0.000000,0.000000,0.000000],[0,0,-1,0],[9E+09,9E+09,9E+09,9E+09,9E+09,9E+09]];
    CONST robtarget T2512:=[[57.999119,79.321798,20.249911],[1.000000,0.000000,0.000000,0.000000],[0,0,-1,0],[9E+09,9E+09,9E+09,9E+09,9E+09,9E+09]];
    CONST robtarget T2513:=[[57.999119,33.369340,20.249911],[1.000000,0.000000,0.000000,0.000000],[0,0,-1,0],[9E+09,9E+09,9E+09,9E+09,9E+09,9E+09]];
    CONST robtarget T2514:=[[59.499125,33.502987,20.249911],[1.000000,0.000000,0.000000,0.000000],[0,0,-1,0],[9E+09,9E+09,9E+09,9E+09,9E+09,9E+09]];
    CONST robtarget T2515:=[[59.499125,78.998069,20.249911],[1.000000,0.000000,0.000000,0.000000],[0,0,-1,0],[9E+09,9E+09,9E+09,9E+09,9E+09,9E+09]];
    CONST robtarget T2516:=[[60.999131,78.607871,20.249911],[1.000000,0.000000,0.000000,0.000000],[0,0,-1,0],[9E+09,9E+09,9E+09,9E+09,9E+09,9E+09]];
    CONST robtarget T2517:=[[60.999131,33.714535,20.249911],[1.000000,0.000000,0.000000,0.000000],[0,0,-1,0],[9E+09,9E+09,9E+09,9E+09,9E+09,9E+09]];
    CONST robtarget T2518:=[[62.499137,33.967477,20.249911],[1.000000,0.000000,0.000000,0.000000],[0,0,-1,0],[9E+09,9E+09,9E+09,9E+09,9E+09,9E+09]];
    CONST robtarget T2519:=[[62.499137,78.046573,20.249911],[1.000000,0.000000,0.000000,0.000000],[0,0,-1,0],[9E+09,9E+09,9E+09,9E+09,9E+09,9E+09]];
    CONST robtarget T2520:=[[63.999143,77.324185,20.249911],[1.000000,0.000000,0.000000,0.000000],[0,0,-1,0],[9E+09,9E+09,9E+09,9E+09,9E+09,9E+09]];
    CONST robtarget T2521:=[[63.999143,34.349893,20.249911],[1.000000,0.000000,0.000000,0.000000],[0,0,-1,0],[9E+09,9E+09,9E+09,9E+09,9E+09,9E+09]];
    CONST robtarget T2522:=[[65.499149,34.782299,20.249911],[1.000000,0.000000,0.000000,0.000000],[0,0,-1,0],[9E+09,9E+09,9E+09,9E+09,9E+09,9E+09]];
    CONST robtarget T2523:=[[65.499149,76.288601,20.249911],[1.000000,0.000000,0.000000,0.000000],[0,0,-1,0],[9E+09,9E+09,9E+09,9E+09,9E+09,9E+09]];
    CONST robtarget T2524:=[[66.999155,74.596967,20.249911],[1.000000,0.000000,0.000000,0.000000],[0,0,-1,0],[9E+09,9E+09,9E+09,9E+09,9E+09,9E+09]];
    CONST robtarget T2525:=[[66.999155,35.383610,20.249911],[1.000000,0.000000,0.000000,0.000000],[0,0,-1,0],[9E+09,9E+09,9E+09,9E+09,9E+09,9E+09]];
    CONST robtarget T2526:=[[68.499161,36.073180,20.249911],[1.000000,0.000000,0.000000,0.000000],[0,0,-1,0],[9E+09,9E+09,9E+09,9E+09,9E+09,9E+09]];
    CONST robtarget T2527:=[[68.499161,72.338240,20.249911],[1.000000,0.000000,0.000000,0.000000],[0,0,-1,0],[9E+09,9E+09,9E+09,9E+09,9E+09,9E+09]];
    CONST robtarget T2528:=[[69.999167,70.369139,20.249911],[1.000000,0.000000,0.000000,0.000000],[0,0,-1,0],[9E+09,9E+09,9E+09,9E+09,9E+09,9E+09]];
    CONST robtarget T2529:=[[69.999167,37.106077,20.249911],[1.000000,0.000000,0.000000,0.000000],[0,0,-1,0],[9E+09,9E+09,9E+09,9E+09,9E+09,9E+09]];
    CONST robtarget T2530:=[[71.499173,38.521920,20.249911],[1.000000,0.000000,0.000000,0.000000],[0,0,-1,0],[9E+09,9E+09,9E+09,9E+09,9E+09,9E+09]];
    CONST robtarget T2531:=[[71.499173,72.382313,20.249911],[1.000000,0.000000,0.000000,0.000000],[0,0,-1,0],[9E+09,9E+09,9E+09,9E+09,9E+09,9E+09]];
    CONST robtarget T2532:=[[72.999179,69.847977,20.249911],[1.000000,0.000000,0.000000,0.000000],[0,0,-1,0],[9E+09,9E+09,9E+09,9E+09,9E+09,9E+09]];
    CONST robtarget T2533:=[[72.999179,40.723946,20.249911],[1.000000,0.000000,0.000000,0.000000],[0,0,-1,0],[9E+09,9E+09,9E+09,9E+09,9E+09,9E+09]];
    CONST robtarget T2534:=[[74.499185,53.922236,20.249911],[1.000000,0.000000,0.000000,0.000000],[0,0,-1,0],[9E+09,9E+09,9E+09,9E+09,9E+09,9E+09]];
    CONST robtarget T2535:=[[74.499185,65.008806,20.249911],[1.000000,0.000000,0.000000,0.000000],[0,0,-1,0],[9E+09,9E+09,9E+09,9E+09,9E+09,9E+09]];
    CONST robtarget T2536:=[[74.497880,57.598568,20.749921],[1.000000,0.000000,0.000000,0.000000],[0,0,-1,0],[9E+09,9E+09,9E+09,9E+09,9E+09,9E+09]];
    CONST robtarget T2537:=[[74.497880,63.498669,20.749921],[1.000000,0.000000,0.000000,0.000000],[0,0,-1,0],[9E+09,9E+09,9E+09,9E+09,9E+09,9E+09]];
    CONST robtarget T2538:=[[74.497880,57.598568,20.749921],[1.000000,0.000000,0.000000,0.000000],[0,0,-1,0],[9E+09,9E+09,9E+09,9E+09,9E+09,9E+09]];
    CONST robtarget T2539:=[[74.497880,63.498669,20.749921],[1.000000,0.000000,0.000000,0.000000],[0,0,-1,0],[9E+09,9E+09,9E+09,9E+09,9E+09,9E+09]];
    CONST robtarget T2540:=[[72.997874,69.290181,20.749921],[1.000000,0.000000,0.000000,0.000000],[0,0,-1,0],[9E+09,9E+09,9E+09,9E+09,9E+09,9E+09]];
    CONST robtarget T2541:=[[72.997874,42.041228,20.749921],[1.000000,0.000000,0.000000,0.000000],[0,0,-1,0],[9E+09,9E+09,9E+09,9E+09,9E+09,9E+09]];
    CONST robtarget T2542:=[[71.497868,39.193273,20.749921],[1.000000,0.000000,0.000000,0.000000],[0,0,-1,0],[9E+09,9E+09,9E+09,9E+09,9E+09,9E+09]];
    CONST robtarget T2543:=[[71.497868,72.277503,20.749921],[1.000000,0.000000,0.000000,0.000000],[0,0,-1,0],[9E+09,9E+09,9E+09,9E+09,9E+09,9E+09]];
    CONST robtarget T2544:=[[69.997862,70.146198,20.749921],[1.000000,0.000000,0.000000,0.000000],[0,0,-1,0],[9E+09,9E+09,9E+09,9E+09,9E+09,9E+09]];
    CONST robtarget T2545:=[[69.997862,37.449444,20.749921],[1.000000,0.000000,0.000000,0.000000],[0,0,-1,0],[9E+09,9E+09,9E+09,9E+09,9E+09,9E+09]];
    CONST robtarget T2546:=[[68.497856,36.338714,20.749921],[1.000000,0.000000,0.000000,0.000000],[0,0,-1,0],[9E+09,9E+09,9E+09,9E+09,9E+09,9E+09]];
    CONST robtarget T2547:=[[68.497856,72.029411,20.749921],[1.000000,0.000000,0.000000,0.000000],[0,0,-1,0],[9E+09,9E+09,9E+09,9E+09,9E+09,9E+09]];
    CONST robtarget T2548:=[[66.997850,74.288823,20.749921],[1.000000,0.000000,0.000000,0.000000],[0,0,-1,0],[9E+09,9E+09,9E+09,9E+09,9E+09,9E+09]];
    CONST robtarget T2549:=[[66.997850,35.608586,20.749921],[1.000000,0.000000,0.000000,0.000000],[0,0,-1,0],[9E+09,9E+09,9E+09,9E+09,9E+09,9E+09]];
    CONST robtarget T2550:=[[65.497844,35.007275,20.749921],[1.000000,0.000000,0.000000,0.000000],[0,0,-1,0],[9E+09,9E+09,9E+09,9E+09,9E+09,9E+09]];
    CONST robtarget T2551:=[[65.497844,76.153765,20.749921],[1.000000,0.000000,0.000000,0.000000],[0,0,-1,0],[9E+09,9E+09,9E+09,9E+09,9E+09,9E+09]];
    CONST robtarget T2552:=[[63.997838,77.232802,20.749921],[1.000000,0.000000,0.000000,0.000000],[0,0,-1,0],[9E+09,9E+09,9E+09,9E+09,9E+09,9E+09]];
    CONST robtarget T2553:=[[63.997838,34.560919,20.749921],[1.000000,0.000000,0.000000,0.000000],[0,0,-1,0],[9E+09,9E+09,9E+09,9E+09,9E+09,9E+09]];
    CONST robtarget T2554:=[[62.497832,34.175427,20.749921],[1.000000,0.000000,0.000000,0.000000],[0,0,-1,0],[9E+09,9E+09,9E+09,9E+09,9E+09,9E+09]];
    CONST robtarget T2555:=[[62.497832,77.964732,20.749921],[1.000000,0.000000,0.000000,0.000000],[0,0,-1,0],[9E+09,9E+09,9E+09,9E+09,9E+09,9E+09]];
    CONST robtarget T2556:=[[60.997826,78.523491,20.749921],[1.000000,0.000000,0.000000,0.000000],[0,0,-1,0],[9E+09,9E+09,9E+09,9E+09,9E+09,9E+09]];
    CONST robtarget T2557:=[[60.997826,33.916660,20.749921],[1.000000,0.000000,0.000000,0.000000],[0,0,-1,0],[9E+09,9E+09,9E+09,9E+09,9E+09,9E+09]];
    CONST robtarget T2558:=[[59.497820,33.705113,20.749921],[1.000000,0.000000,0.000000,0.000000],[0,0,-1,0],[9E+09,9E+09,9E+09,9E+09,9E+09,9E+09]];
    CONST robtarget T2559:=[[59.497820,78.914680,20.749921],[1.000000,0.000000,0.000000,0.000000],[0,0,-1,0],[9E+09,9E+09,9E+09,9E+09,9E+09,9E+09]];
    CONST robtarget T2560:=[[57.997814,79.252099,20.749921],[1.000000,0.000000,0.000000,0.000000],[0,0,-1,0],[9E+09,9E+09,9E+09,9E+09,9E+09,9E+09]];
    CONST robtarget T2561:=[[57.997814,33.569304,20.749921],[1.000000,0.000000,0.000000,0.000000],[0,0,-1,0],[9E+09,9E+09,9E+09,9E+09,9E+09,9E+09]];
    CONST robtarget T2562:=[[56.497808,33.470027,20.749921],[1.000000,0.000000,0.000000,0.000000],[0,0,-1,0],[9E+09,9E+09,9E+09,9E+09,9E+09,9E+09]];
    CONST robtarget T2563:=[[56.497808,79.597417,20.749921],[1.000000,0.000000,0.000000,0.000000],[0,0,-1,0],[9E+09,9E+09,9E+09,9E+09,9E+09,9E+09]];
    CONST robtarget T2564:=[[54.997802,79.856688,20.749921],[1.000000,0.000000,0.000000,0.000000],[0,0,-1,0],[9E+09,9E+09,9E+09,9E+09,9E+09,9E+09]];
    CONST robtarget T2565:=[[54.997802,33.453294,20.749921],[1.000000,0.000000,0.000000,0.000000],[0,0,-1,0],[9E+09,9E+09,9E+09,9E+09,9E+09,9E+09]];
    CONST robtarget T2566:=[[53.497796,33.470151,20.749921],[1.000000,0.000000,0.000000,0.000000],[0,0,-1,0],[9E+09,9E+09,9E+09,9E+09,9E+09,9E+09]];
    CONST robtarget T2567:=[[53.497796,79.596259,20.749921],[1.000000,0.000000,0.000000,0.000000],[0,0,-1,0],[9E+09,9E+09,9E+09,9E+09,9E+09,9E+09]];
    CONST robtarget T2568:=[[51.997790,79.251179,20.749921],[1.000000,0.000000,0.000000,0.000000],[0,0,-1,0],[9E+09,9E+09,9E+09,9E+09,9E+09,9E+09]];
    CONST robtarget T2569:=[[51.997790,33.569669,20.749921],[1.000000,0.000000,0.000000,0.000000],[0,0,-1,0],[9E+09,9E+09,9E+09,9E+09,9E+09,9E+09]];
    CONST robtarget T2570:=[[50.497784,33.705735,20.749921],[1.000000,0.000000,0.000000,0.000000],[0,0,-1,0],[9E+09,9E+09,9E+09,9E+09,9E+09,9E+09]];
    CONST robtarget T2571:=[[50.497784,78.913578,20.749921],[1.000000,0.000000,0.000000,0.000000],[0,0,-1,0],[9E+09,9E+09,9E+09,9E+09,9E+09,9E+09]];
    CONST robtarget T2572:=[[48.997778,78.522035,20.749921],[1.000000,0.000000,0.000000,0.000000],[0,0,-1,0],[9E+09,9E+09,9E+09,9E+09,9E+09,9E+09]];
    CONST robtarget T2573:=[[48.997778,33.917282,20.749921],[1.000000,0.000000,0.000000,0.000000],[0,0,-1,0],[9E+09,9E+09,9E+09,9E+09,9E+09,9E+09]];
    CONST robtarget T2574:=[[47.497772,34.176537,20.749921],[1.000000,0.000000,0.000000,0.000000],[0,0,-1,0],[9E+09,9E+09,9E+09,9E+09,9E+09,9E+09]];
    CONST robtarget T2575:=[[47.497772,77.963073,20.749921],[1.000000,0.000000,0.000000,0.000000],[0,0,-1,0],[9E+09,9E+09,9E+09,9E+09,9E+09,9E+09]];
    CONST robtarget T2576:=[[45.997766,77.230746,20.749921],[1.000000,0.000000,0.000000,0.000000],[0,0,-1,0],[9E+09,9E+09,9E+09,9E+09,9E+09,9E+09]];
    CONST robtarget T2577:=[[45.997766,34.562057,20.749921],[1.000000,0.000000,0.000000,0.000000],[0,0,-1,0],[9E+09,9E+09,9E+09,9E+09,9E+09,9E+09]];
    CONST robtarget T2578:=[[44.497760,35.009043,20.749921],[1.000000,0.000000,0.000000,0.000000],[0,0,-1,0],[9E+09,9E+09,9E+09,9E+09,9E+09,9E+09]];
    CONST robtarget T2579:=[[44.497760,76.150321,20.749921],[1.000000,0.000000,0.000000,0.000000],[0,0,-1,0],[9E+09,9E+09,9E+09,9E+09,9E+09,9E+09]];
    CONST robtarget T2580:=[[42.997754,74.281416,20.749921],[1.000000,0.000000,0.000000,0.000000],[0,0,-1,0],[9E+09,9E+09,9E+09,9E+09,9E+09,9E+09]];
    CONST robtarget T2581:=[[42.997754,35.610354,20.749921],[1.000000,0.000000,0.000000,0.000000],[0,0,-1,0],[9E+09,9E+09,9E+09,9E+09,9E+09,9E+09]];
    CONST robtarget T2582:=[[41.497748,36.341772,20.749921],[1.000000,0.000000,0.000000,0.000000],[0,0,-1,0],[9E+09,9E+09,9E+09,9E+09,9E+09,9E+09]];
    CONST robtarget T2583:=[[41.497748,72.023043,20.749921],[1.000000,0.000000,0.000000,0.000000],[0,0,-1,0],[9E+09,9E+09,9E+09,9E+09,9E+09,9E+09]];
    CONST robtarget T2584:=[[39.997742,70.141984,20.749921],[1.000000,0.000000,0.000000,0.000000],[0,0,-1,0],[9E+09,9E+09,9E+09,9E+09,9E+09,9E+09]];
    CONST robtarget T2585:=[[39.997742,37.452747,20.749921],[1.000000,0.000000,0.000000,0.000000],[0,0,-1,0],[9E+09,9E+09,9E+09,9E+09,9E+09,9E+09]];
    CONST robtarget T2586:=[[38.497736,39.199629,20.749921],[1.000000,0.000000,0.000000,0.000000],[0,0,-1,0],[9E+09,9E+09,9E+09,9E+09,9E+09,9E+09]];
    CONST robtarget T2587:=[[38.497736,72.272753,20.749921],[1.000000,0.000000,0.000000,0.000000],[0,0,-1,0],[9E+09,9E+09,9E+09,9E+09,9E+09,9E+09]];
    CONST robtarget T2588:=[[36.997730,69.277263,20.749921],[1.000000,0.000000,0.000000,0.000000],[0,0,-1,0],[9E+09,9E+09,9E+09,9E+09,9E+09,9E+09]];
    CONST robtarget T2589:=[[36.997730,42.052764,20.749921],[1.000000,0.000000,0.000000,0.000000],[0,0,-1,0],[9E+09,9E+09,9E+09,9E+09,9E+09,9E+09]];
    CONST robtarget T2590:=[[35.497724,57.602880,20.749921],[1.000000,0.000000,0.000000,0.000000],[0,0,-1,0],[9E+09,9E+09,9E+09,9E+09,9E+09,9E+09]];
    CONST robtarget T2591:=[[35.497724,63.459901,20.749921],[1.000000,0.000000,0.000000,0.000000],[0,0,-1,0],[9E+09,9E+09,9E+09,9E+09,9E+09,9E+09]];
    CONST robtarget T2592:=[[36.243115,58.828178,21.249931],[1.000000,0.000000,0.000000,0.000000],[0,0,-1,0],[9E+09,9E+09,9E+09,9E+09,9E+09,9E+09]];
    CONST robtarget T2593:=[[36.243115,65.536186,21.249931],[1.000000,0.000000,0.000000,0.000000],[0,0,-1,0],[9E+09,9E+09,9E+09,9E+09,9E+09,9E+09]];
    CONST robtarget T2594:=[[36.243115,58.828178,21.249931],[1.000000,0.000000,0.000000,0.000000],[0,0,-1,0],[9E+09,9E+09,9E+09,9E+09,9E+09,9E+09]];
    CONST robtarget T2595:=[[36.243115,65.536186,21.249931],[1.000000,0.000000,0.000000,0.000000],[0,0,-1,0],[9E+09,9E+09,9E+09,9E+09,9E+09,9E+09]];
    CONST robtarget T2596:=[[37.743121,70.537383,21.249931],[1.000000,0.000000,0.000000,0.000000],[0,0,-1,0],[9E+09,9E+09,9E+09,9E+09,9E+09,9E+09]];
    CONST robtarget T2597:=[[37.743121,41.369634,21.249931],[1.000000,0.000000,0.000000,0.000000],[0,0,-1,0],[9E+09,9E+09,9E+09,9E+09,9E+09,9E+09]];
    CONST robtarget T2598:=[[39.243127,38.910455,21.249931],[1.000000,0.000000,0.000000,0.000000],[0,0,-1,0],[9E+09,9E+09,9E+09,9E+09,9E+09,9E+09]];
    CONST robtarget T2599:=[[39.243127,72.646224,21.249931],[1.000000,0.000000,0.000000,0.000000],[0,0,-1,0],[9E+09,9E+09,9E+09,9E+09,9E+09,9E+09]];
    CONST robtarget T2600:=[[40.743133,70.478269,21.249931],[1.000000,0.000000,0.000000,0.000000],[0,0,-1,0],[9E+09,9E+09,9E+09,9E+09,9E+09,9E+09]];
    CONST robtarget T2601:=[[40.743133,37.414042,21.249931],[1.000000,0.000000,0.000000,0.000000],[0,0,-1,0],[9E+09,9E+09,9E+09,9E+09,9E+09,9E+09]];
    CONST robtarget T2602:=[[42.243139,36.299529,21.249931],[1.000000,0.000000,0.000000,0.000000],[0,0,-1,0],[9E+09,9E+09,9E+09,9E+09,9E+09,9E+09]];
    CONST robtarget T2603:=[[42.243139,72.787274,21.249931],[1.000000,0.000000,0.000000,0.000000],[0,0,-1,0],[9E+09,9E+09,9E+09,9E+09,9E+09,9E+09]];
    CONST robtarget T2604:=[[43.743145,75.100102,21.249931],[1.000000,0.000000,0.000000,0.000000],[0,0,-1,0],[9E+09,9E+09,9E+09,9E+09,9E+09,9E+09]];
    CONST robtarget T2605:=[[43.743145,35.625222,21.249931],[1.000000,0.000000,0.000000,0.000000],[0,0,-1,0],[9E+09,9E+09,9E+09,9E+09,9E+09,9E+09]];
    CONST robtarget T2606:=[[45.243151,34.969356,21.249931],[1.000000,0.000000,0.000000,0.000000],[0,0,-1,0],[9E+09,9E+09,9E+09,9E+09,9E+09,9E+09]];
    CONST robtarget T2607:=[[45.243151,76.599714,21.249931],[1.000000,0.000000,0.000000,0.000000],[0,0,-1,0],[9E+09,9E+09,9E+09,9E+09,9E+09,9E+09]];
    CONST robtarget T2608:=[[46.743157,77.503014,21.249931],[1.000000,0.000000,0.000000,0.000000],[0,0,-1,0],[9E+09,9E+09,9E+09,9E+09,9E+09,9E+09]];
    CONST robtarget T2609:=[[46.743157,34.581083,21.249931],[1.000000,0.000000,0.000000,0.000000],[0,0,-1,0],[9E+09,9E+09,9E+09,9E+09,9E+09,9E+09]];
    CONST robtarget T2610:=[[48.243163,34.226016,21.249931],[1.000000,0.000000,0.000000,0.000000],[0,0,-1,0],[9E+09,9E+09,9E+09,9E+09,9E+09,9E+09]];
    CONST robtarget T2611:=[[48.243163,78.159669,21.249931],[1.000000,0.000000,0.000000,0.000000],[0,0,-1,0],[9E+09,9E+09,9E+09,9E+09,9E+09,9E+09]];
    CONST robtarget T2612:=[[49.743169,78.642967,21.249931],[1.000000,0.000000,0.000000,0.000000],[0,0,-1,0],[9E+09,9E+09,9E+09,9E+09,9E+09,9E+09]];
    CONST robtarget T2613:=[[49.743169,34.014469,21.249931],[1.000000,0.000000,0.000000,0.000000],[0,0,-1,0],[9E+09,9E+09,9E+09,9E+09,9E+09,9E+09]];
    CONST robtarget T2614:=[[51.243175,33.831351,21.249931],[1.000000,0.000000,0.000000,0.000000],[0,0,-1,0],[9E+09,9E+09,9E+09,9E+09,9E+09,9E+09]];
    CONST robtarget T2615:=[[51.243175,79.013723,21.249931],[1.000000,0.000000,0.000000,0.000000],[0,0,-1,0],[9E+09,9E+09,9E+09,9E+09,9E+09,9E+09]];
    CONST robtarget T2616:=[[52.743181,79.315819,21.249931],[1.000000,0.000000,0.000000,0.000000],[0,0,-1,0],[9E+09,9E+09,9E+09,9E+09,9E+09,9E+09]];
    CONST robtarget T2617:=[[52.743181,33.706265,21.249931],[1.000000,0.000000,0.000000,0.000000],[0,0,-1,0],[9E+09,9E+09,9E+09,9E+09,9E+09,9E+09]];
    CONST robtarget T2618:=[[54.243187,33.664494,21.249931],[1.000000,0.000000,0.000000,0.000000],[0,0,-1,0],[9E+09,9E+09,9E+09,9E+09,9E+09,9E+09]];
    CONST robtarget T2619:=[[54.243187,79.668490,21.249931],[1.000000,0.000000,0.000000,0.000000],[0,0,-1,0],[9E+09,9E+09,9E+09,9E+09,9E+09,9E+09]];
    CONST robtarget T2620:=[[55.743193,79.670680,21.249931],[1.000000,0.000000,0.000000,0.000000],[0,0,-1,0],[9E+09,9E+09,9E+09,9E+09,9E+09,9E+09]];
    CONST robtarget T2621:=[[55.743193,33.664381,21.249931],[1.000000,0.000000,0.000000,0.000000],[0,0,-1,0],[9E+09,9E+09,9E+09,9E+09,9E+09,9E+09]];
    CONST robtarget T2622:=[[57.243199,33.705071,21.249931],[1.000000,0.000000,0.000000,0.000000],[0,0,-1,0],[9E+09,9E+09,9E+09,9E+09,9E+09,9E+09]];
    CONST robtarget T2623:=[[57.243199,79.318087,21.249931],[1.000000,0.000000,0.000000,0.000000],[0,0,-1,0],[9E+09,9E+09,9E+09,9E+09,9E+09,9E+09]];
    CONST robtarget T2624:=[[58.743205,79.016544,21.249931],[1.000000,0.000000,0.000000,0.000000],[0,0,-1,0],[9E+09,9E+09,9E+09,9E+09,9E+09,9E+09]];
    CONST robtarget T2625:=[[58.743205,33.830223,21.249931],[1.000000,0.000000,0.000000,0.000000],[0,0,-1,0],[9E+09,9E+09,9E+09,9E+09,9E+09,9E+09]];
    CONST robtarget T2626:=[[60.243211,34.012546,21.249931],[1.000000,0.000000,0.000000,0.000000],[0,0,-1,0],[9E+09,9E+09,9E+09,9E+09,9E+09,9E+09]];
    CONST robtarget T2627:=[[60.243211,78.646082,21.249931],[1.000000,0.000000,0.000000,0.000000],[0,0,-1,0],[9E+09,9E+09,9E+09,9E+09,9E+09,9E+09]];
    CONST robtarget T2628:=[[61.743217,78.164778,21.249931],[1.000000,0.000000,0.000000,0.000000],[0,0,-1,0],[9E+09,9E+09,9E+09,9E+09,9E+09,9E+09]];
    CONST robtarget T2629:=[[61.743217,34.224093,21.249931],[1.000000,0.000000,0.000000,0.000000],[0,0,-1,0],[9E+09,9E+09,9E+09,9E+09,9E+09,9E+09]];
    CONST robtarget T2630:=[[63.243223,34.577565,21.249931],[1.000000,0.000000,0.000000,0.000000],[0,0,-1,0],[9E+09,9E+09,9E+09,9E+09,9E+09,9E+09]];
    CONST robtarget T2631:=[[63.243223,77.509853,21.249931],[1.000000,0.000000,0.000000,0.000000],[0,0,-1,0],[9E+09,9E+09,9E+09,9E+09,9E+09,9E+09]];
    CONST robtarget T2632:=[[64.743229,76.610988,21.249931],[1.000000,0.000000,0.000000,0.000000],[0,0,-1,0],[9E+09,9E+09,9E+09,9E+09,9E+09,9E+09]];
    CONST robtarget T2633:=[[64.743229,34.965284,21.249931],[1.000000,0.000000,0.000000,0.000000],[0,0,-1,0],[9E+09,9E+09,9E+09,9E+09,9E+09,9E+09]];
    CONST robtarget T2634:=[[66.243235,35.618942,21.249931],[1.000000,0.000000,0.000000,0.000000],[0,0,-1,0],[9E+09,9E+09,9E+09,9E+09,9E+09,9E+09]];
    CONST robtarget T2635:=[[66.243235,75.118669,21.249931],[1.000000,0.000000,0.000000,0.000000],[0,0,-1,0],[9E+09,9E+09,9E+09,9E+09,9E+09,9E+09]];
    CONST robtarget T2636:=[[67.743241,72.806803,21.249931],[1.000000,0.000000,0.000000,0.000000],[0,0,-1,0],[9E+09,9E+09,9E+09,9E+09,9E+09,9E+09]];
    CONST robtarget T2637:=[[67.743241,36.290381,21.249931],[1.000000,0.000000,0.000000,0.000000],[0,0,-1,0],[9E+09,9E+09,9E+09,9E+09,9E+09,9E+09]];
    CONST robtarget T2638:=[[69.243247,37.403830,21.249931],[1.000000,0.000000,0.000000,0.000000],[0,0,-1,0],[9E+09,9E+09,9E+09,9E+09,9E+09,9E+09]];
    CONST robtarget T2639:=[[69.243247,70.499973,21.249931],[1.000000,0.000000,0.000000,0.000000],[0,0,-1,0],[9E+09,9E+09,9E+09,9E+09,9E+09,9E+09]];
    CONST robtarget T2640:=[[70.743253,72.649823,21.249931],[1.000000,0.000000,0.000000,0.000000],[0,0,-1,0],[9E+09,9E+09,9E+09,9E+09,9E+09,9E+09]];
    CONST robtarget T2641:=[[70.743253,38.890799,21.249931],[1.000000,0.000000,0.000000,0.000000],[0,0,-1,0],[9E+09,9E+09,9E+09,9E+09,9E+09,9E+09]];
    CONST robtarget T2642:=[[72.243259,41.330876,21.249931],[1.000000,0.000000,0.000000,0.000000],[0,0,-1,0],[9E+09,9E+09,9E+09,9E+09,9E+09,9E+09]];
    CONST robtarget T2643:=[[72.243259,70.564142,21.249931],[1.000000,0.000000,0.000000,0.000000],[0,0,-1,0],[9E+09,9E+09,9E+09,9E+09,9E+09,9E+09]];
    CONST robtarget T2644:=[[73.743265,65.604666,21.249931],[1.000000,0.000000,0.000000,0.000000],[0,0,-1,0],[9E+09,9E+09,9E+09,9E+09,9E+09,9E+09]];
    CONST robtarget T2645:=[[73.743265,58.832518,21.249931],[1.000000,0.000000,0.000000,0.000000],[0,0,-1,0],[9E+09,9E+09,9E+09,9E+09,9E+09,9E+09]];
    CONST robtarget T2646:=[[72.988108,60.829353,21.749941],[1.000000,0.000000,0.000000,0.000000],[0,0,-1,0],[9E+09,9E+09,9E+09,9E+09,9E+09,9E+09]];
    CONST robtarget T2647:=[[72.988108,67.598939,21.749941],[1.000000,0.000000,0.000000,0.000000],[0,0,-1,0],[9E+09,9E+09,9E+09,9E+09,9E+09,9E+09]];
    CONST robtarget T2648:=[[72.988108,60.829353,21.749941],[1.000000,0.000000,0.000000,0.000000],[0,0,-1,0],[9E+09,9E+09,9E+09,9E+09,9E+09,9E+09]];
    CONST robtarget T2649:=[[72.988108,67.598939,21.749941],[1.000000,0.000000,0.000000,0.000000],[0,0,-1,0],[9E+09,9E+09,9E+09,9E+09,9E+09,9E+09]];
    CONST robtarget T2650:=[[71.488102,71.631499,21.749941],[1.000000,0.000000,0.000000,0.000000],[0,0,-1,0],[9E+09,9E+09,9E+09,9E+09,9E+09,9E+09]];
    CONST robtarget T2651:=[[71.488102,64.340248,21.749941],[1.000000,0.000000,0.000000,0.000000],[0,0,-1,0],[9E+09,9E+09,9E+09,9E+09,9E+09,9E+09]];
    CONST robtarget T2652:=[[71.488102,63.102045,21.749941],[1.000000,0.000000,0.000000,0.000000],[0,0,-1,0],[9E+09,9E+09,9E+09,9E+09,9E+09,9E+09]];
    CONST robtarget T2653:=[[71.488102,40.769853,21.749941],[1.000000,0.000000,0.000000,0.000000],[0,0,-1,0],[9E+09,9E+09,9E+09,9E+09,9E+09,9E+09]];
    CONST robtarget T2654:=[[69.988096,38.587545,21.749941],[1.000000,0.000000,0.000000,0.000000],[0,0,-1,0],[9E+09,9E+09,9E+09,9E+09,9E+09,9E+09]];
    CONST robtarget T2655:=[[69.988096,68.686094,21.749941],[1.000000,0.000000,0.000000,0.000000],[0,0,-1,0],[9E+09,9E+09,9E+09,9E+09,9E+09,9E+09]];
    CONST robtarget T2656:=[[69.988096,69.635370,21.749941],[1.000000,0.000000,0.000000,0.000000],[0,0,-1,0],[9E+09,9E+09,9E+09,9E+09,9E+09,9E+09]];
    CONST robtarget T2657:=[[69.988096,72.390587,21.749941],[1.000000,0.000000,0.000000,0.000000],[0,0,-1,0],[9E+09,9E+09,9E+09,9E+09,9E+09,9E+09]];
    CONST robtarget T2658:=[[68.488090,71.335749,21.749941],[1.000000,0.000000,0.000000,0.000000],[0,0,-1,0],[9E+09,9E+09,9E+09,9E+09,9E+09,9E+09]];
    CONST robtarget T2659:=[[68.488090,37.357810,21.749941],[1.000000,0.000000,0.000000,0.000000],[0,0,-1,0],[9E+09,9E+09,9E+09,9E+09,9E+09,9E+09]];
    CONST robtarget T2660:=[[66.988084,36.398170,21.749941],[1.000000,0.000000,0.000000,0.000000],[0,0,-1,0],[9E+09,9E+09,9E+09,9E+09,9E+09,9E+09]];
    CONST robtarget T2661:=[[66.988084,73.684557,21.749941],[1.000000,0.000000,0.000000,0.000000],[0,0,-1,0],[9E+09,9E+09,9E+09,9E+09,9E+09,9E+09]];
    CONST robtarget T2662:=[[65.488078,75.830385,21.749941],[1.000000,0.000000,0.000000,0.000000],[0,0,-1,0],[9E+09,9E+09,9E+09,9E+09,9E+09,9E+09]];
    CONST robtarget T2663:=[[65.488078,35.726940,21.749941],[1.000000,0.000000,0.000000,0.000000],[0,0,-1,0],[9E+09,9E+09,9E+09,9E+09,9E+09,9E+09]];
    CONST robtarget T2664:=[[63.988072,35.147369,21.749941],[1.000000,0.000000,0.000000,0.000000],[0,0,-1,0],[9E+09,9E+09,9E+09,9E+09,9E+09,9E+09]];
    CONST robtarget T2665:=[[63.988072,77.064332,21.749941],[1.000000,0.000000,0.000000,0.000000],[0,0,-1,0],[9E+09,9E+09,9E+09,9E+09,9E+09,9E+09]];
    CONST robtarget T2666:=[[62.488066,77.791803,21.749941],[1.000000,0.000000,0.000000,0.000000],[0,0,-1,0],[9E+09,9E+09,9E+09,9E+09,9E+09,9E+09]];
    CONST robtarget T2667:=[[62.488066,34.699453,21.749941],[1.000000,0.000000,0.000000,0.000000],[0,0,-1,0],[9E+09,9E+09,9E+09,9E+09,9E+09,9E+09]];
    CONST robtarget T2668:=[[60.988060,34.355613,21.749941],[1.000000,0.000000,0.000000,0.000000],[0,0,-1,0],[9E+09,9E+09,9E+09,9E+09,9E+09,9E+09]];
    CONST robtarget T2669:=[[60.988060,78.352434,21.749941],[1.000000,0.000000,0.000000,0.000000],[0,0,-1,0],[9E+09,9E+09,9E+09,9E+09,9E+09,9E+09]];
    CONST robtarget T2670:=[[59.488054,78.749687,21.749941],[1.000000,0.000000,0.000000,0.000000],[0,0,-1,0],[9E+09,9E+09,9E+09,9E+09,9E+09,9E+09]];
    CONST robtarget T2671:=[[59.488054,34.108355,21.749941],[1.000000,0.000000,0.000000,0.000000],[0,0,-1,0],[9E+09,9E+09,9E+09,9E+09,9E+09,9E+09]];
    CONST robtarget T2672:=[[57.988048,33.967067,21.749941],[1.000000,0.000000,0.000000,0.000000],[0,0,-1,0],[9E+09,9E+09,9E+09,9E+09,9E+09,9E+09]];
    CONST robtarget T2673:=[[57.988048,79.091394,21.749941],[1.000000,0.000000,0.000000,0.000000],[0,0,-1,0],[9E+09,9E+09,9E+09,9E+09,9E+09,9E+09]];
    CONST robtarget T2674:=[[56.488042,79.409586,21.749941],[1.000000,0.000000,0.000000,0.000000],[0,0,-1,0],[9E+09,9E+09,9E+09,9E+09,9E+09,9E+09]];
    CONST robtarget T2675:=[[56.488042,33.875500,21.749941],[1.000000,0.000000,0.000000,0.000000],[0,0,-1,0],[9E+09,9E+09,9E+09,9E+09,9E+09,9E+09]];
    CONST robtarget T2676:=[[54.988036,33.863310,21.749941],[1.000000,0.000000,0.000000,0.000000],[0,0,-1,0],[9E+09,9E+09,9E+09,9E+09,9E+09,9E+09]];
    CONST robtarget T2677:=[[54.988036,79.686562,21.749941],[1.000000,0.000000,0.000000,0.000000],[0,0,-1,0],[9E+09,9E+09,9E+09,9E+09,9E+09,9E+09]];
    CONST robtarget T2678:=[[53.488030,79.403328,21.749941],[1.000000,0.000000,0.000000,0.000000],[0,0,-1,0],[9E+09,9E+09,9E+09,9E+09,9E+09,9E+09]];
    CONST robtarget T2679:=[[53.488030,33.875698,21.749941],[1.000000,0.000000,0.000000,0.000000],[0,0,-1,0],[9E+09,9E+09,9E+09,9E+09,9E+09,9E+09]];
    CONST robtarget T2680:=[[51.988024,33.969047,21.749941],[1.000000,0.000000,0.000000,0.000000],[0,0,-1,0],[9E+09,9E+09,9E+09,9E+09,9E+09,9E+09]];
    CONST robtarget T2681:=[[51.988024,79.086435,21.749941],[1.000000,0.000000,0.000000,0.000000],[0,0,-1,0],[9E+09,9E+09,9E+09,9E+09,9E+09,9E+09]];
    CONST robtarget T2682:=[[50.488018,78.743716,21.749941],[1.000000,0.000000,0.000000,0.000000],[0,0,-1,0],[9E+09,9E+09,9E+09,9E+09,9E+09,9E+09]];
    CONST robtarget T2683:=[[50.488018,34.111732,21.749941],[1.000000,0.000000,0.000000,0.000000],[0,0,-1,0],[9E+09,9E+09,9E+09,9E+09,9E+09,9E+09]];
    CONST robtarget T2684:=[[48.988012,34.359836,21.749941],[1.000000,0.000000,0.000000,0.000000],[0,0,-1,0],[9E+09,9E+09,9E+09,9E+09,9E+09,9E+09]];
    CONST robtarget T2685:=[[48.988012,78.344564,21.749941],[1.000000,0.000000,0.000000,0.000000],[0,0,-1,0],[9E+09,9E+09,9E+09,9E+09,9E+09,9E+09]];
    CONST robtarget T2686:=[[47.488006,77.779792,21.749941],[1.000000,0.000000,0.000000,0.000000],[0,0,-1,0],[9E+09,9E+09,9E+09,9E+09,9E+09,9E+09]];
    CONST robtarget T2687:=[[47.488006,34.706603,21.749941],[1.000000,0.000000,0.000000,0.000000],[0,0,-1,0],[9E+09,9E+09,9E+09,9E+09,9E+09,9E+09]];
    CONST robtarget T2688:=[[45.988000,35.154519,21.749941],[1.000000,0.000000,0.000000,0.000000],[0,0,-1,0],[9E+09,9E+09,9E+09,9E+09,9E+09,9E+09]];
    CONST robtarget T2689:=[[45.988000,77.053177,21.749941],[1.000000,0.000000,0.000000,0.000000],[0,0,-1,0],[9E+09,9E+09,9E+09,9E+09,9E+09,9E+09]];
    CONST robtarget T2690:=[[44.487994,75.802674,21.749941],[1.000000,0.000000,0.000000,0.000000],[0,0,-1,0],[9E+09,9E+09,9E+09,9E+09,9E+09,9E+09]];
    CONST robtarget T2691:=[[44.487994,35.737968,21.749941],[1.000000,0.000000,0.000000,0.000000],[0,0,-1,0],[9E+09,9E+09,9E+09,9E+09,9E+09,9E+09]];
    CONST robtarget T2692:=[[42.987988,36.407874,21.749941],[1.000000,0.000000,0.000000,0.000000],[0,0,-1,0],[9E+09,9E+09,9E+09,9E+09,9E+09,9E+09]];
    CONST robtarget T2693:=[[42.987988,73.644332,21.749941],[1.000000,0.000000,0.000000,0.000000],[0,0,-1,0],[9E+09,9E+09,9E+09,9E+09,9E+09,9E+09]];
    CONST robtarget T2694:=[[41.487982,71.297592,21.749941],[1.000000,0.000000,0.000000,0.000000],[0,0,-1,0],[9E+09,9E+09,9E+09,9E+09,9E+09,9E+09]];
